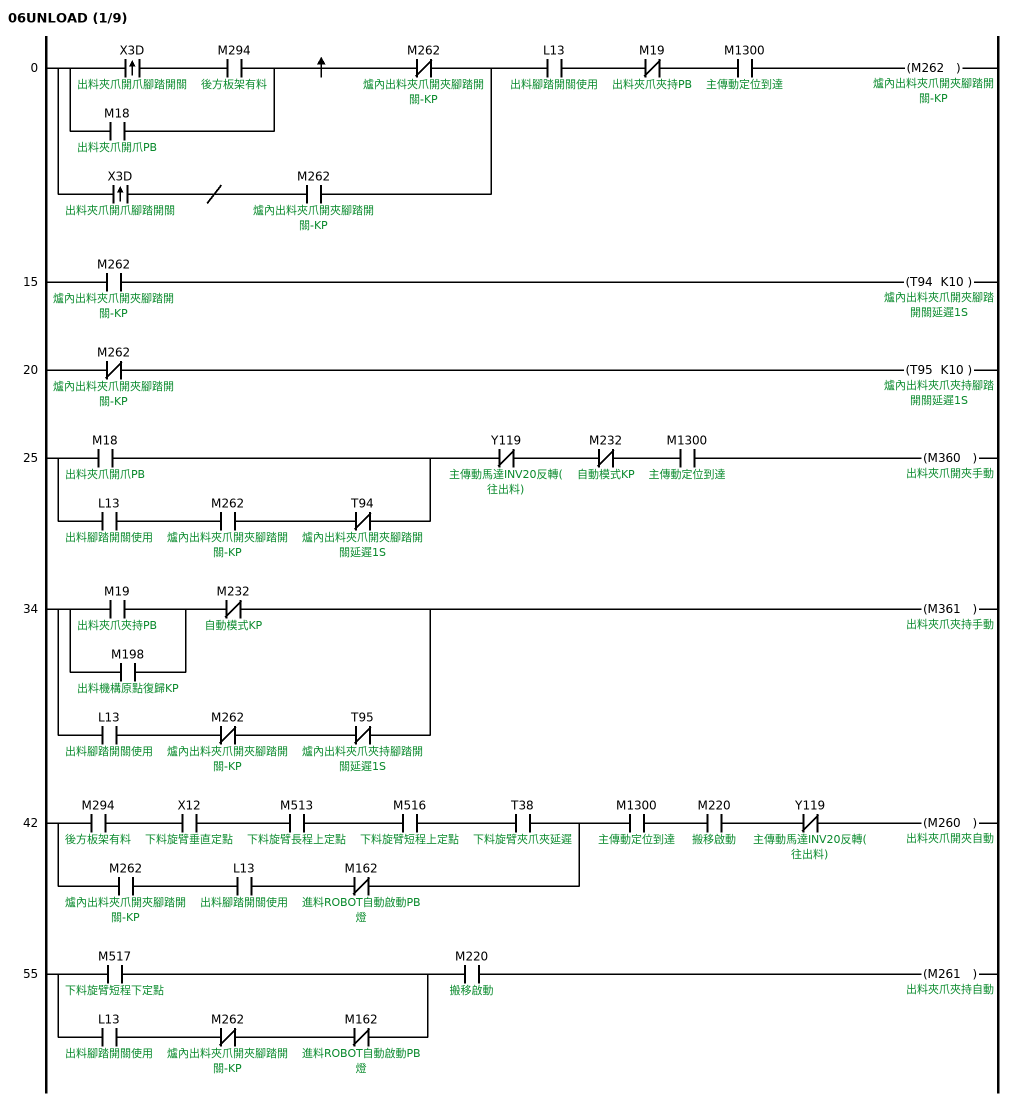
[picture p24: ladder of 06UNLOAD, rungs at steps 0 to 55]
0     LDP     X3D  ; 出料夾爪開爪腳踏開關
      AND     M294  ; 後方板架有料
      OR      M18  ; 出料夾爪開爪PB
      MEP
      ANI     M262  ; 爐內出料夾爪開夾腳踏開關-KP
      LDP     X3D  ; 出料夾爪開爪腳踏開關
      INV
      AND     M262  ; 爐內出料夾爪開夾腳踏開關-KP
      ORB
      AND     L13  ; 出料腳踏開關使用
      ANI     M19  ; 出料夾爪夾持PB
      AND     M1300  ; 主傳動定位到達
      OUT     M262  ; 爐內出料夾爪開夾腳踏開關-KP
15    LD      M262  ; 爐內出料夾爪開夾腳踏開關-KP
      OUT     T94 K10  ; 爐內出料夾爪開夾腳踏開關延遲1S
20    LDI     M262  ; 爐內出料夾爪開夾腳踏開關-KP
      OUT     T95 K10  ; 爐內出料夾爪夾持腳踏開關延遲1S
25    LD      M18  ; 出料夾爪開爪PB
      LD      L13  ; 出料腳踏開關使用
      AND     M262  ; 爐內出料夾爪開夾腳踏開關-KP
      ANI     T94  ; 爐內出料夾爪開夾腳踏開關延遲1S
      ORB
      ANI     Y119  ; 主傳動馬達INV20反轉(往出料)
      ANI     M232  ; 自動模式KP
      AND     M1300  ; 主傳動定位到達
      OUT     M360  ; 出料夾爪開夾手動
34    LD      M19  ; 出料夾爪夾持PB
      OR      M198  ; 出料機構原點復歸KP
      ANI     M232  ; 自動模式KP
      LD      L13  ; 出料腳踏開關使用
      ANI     M262  ; 爐內出料夾爪開夾腳踏開關-KP
      ANI     T95  ; 爐內出料夾爪夾持腳踏開關延遲1S
      ORB
      OUT     M361  ; 出料夾爪夾持手動
42    LD      M294  ; 後方板架有料
      AND     X12  ; 下料旋臂垂直定點
      AND     M513  ; 下料旋臂長程上定點
      AND     M516  ; 下料旋臂短程上定點
      AND     T38  ; 下料旋臂夾爪夾延遲
      LD      M262  ; 爐內出料夾爪開夾腳踏開關-KP
      AND     L13  ; 出料腳踏開關使用
      ANI     M162  ; 進料ROBOT自動啟動PB燈
      ORB
      AND     M1300  ; 主傳動定位到達
      AND     M220  ; 搬移啟動
      ANI     Y119  ; 主傳動馬達INV20反轉(往出料)
      OUT     M260  ; 出料夾爪開夾自動
55    LD      M517  ; 下料旋臂短程下定點
      LD      L13  ; 出料腳踏開關使用
      ANI     M262  ; 爐內出料夾爪開夾腳踏開關-KP
      ANI     M162  ; 進料ROBOT自動啟動PB燈
      ORB
      AND     M220  ; 搬移啟動
      OUT     M261  ; 出料夾爪夾持自動
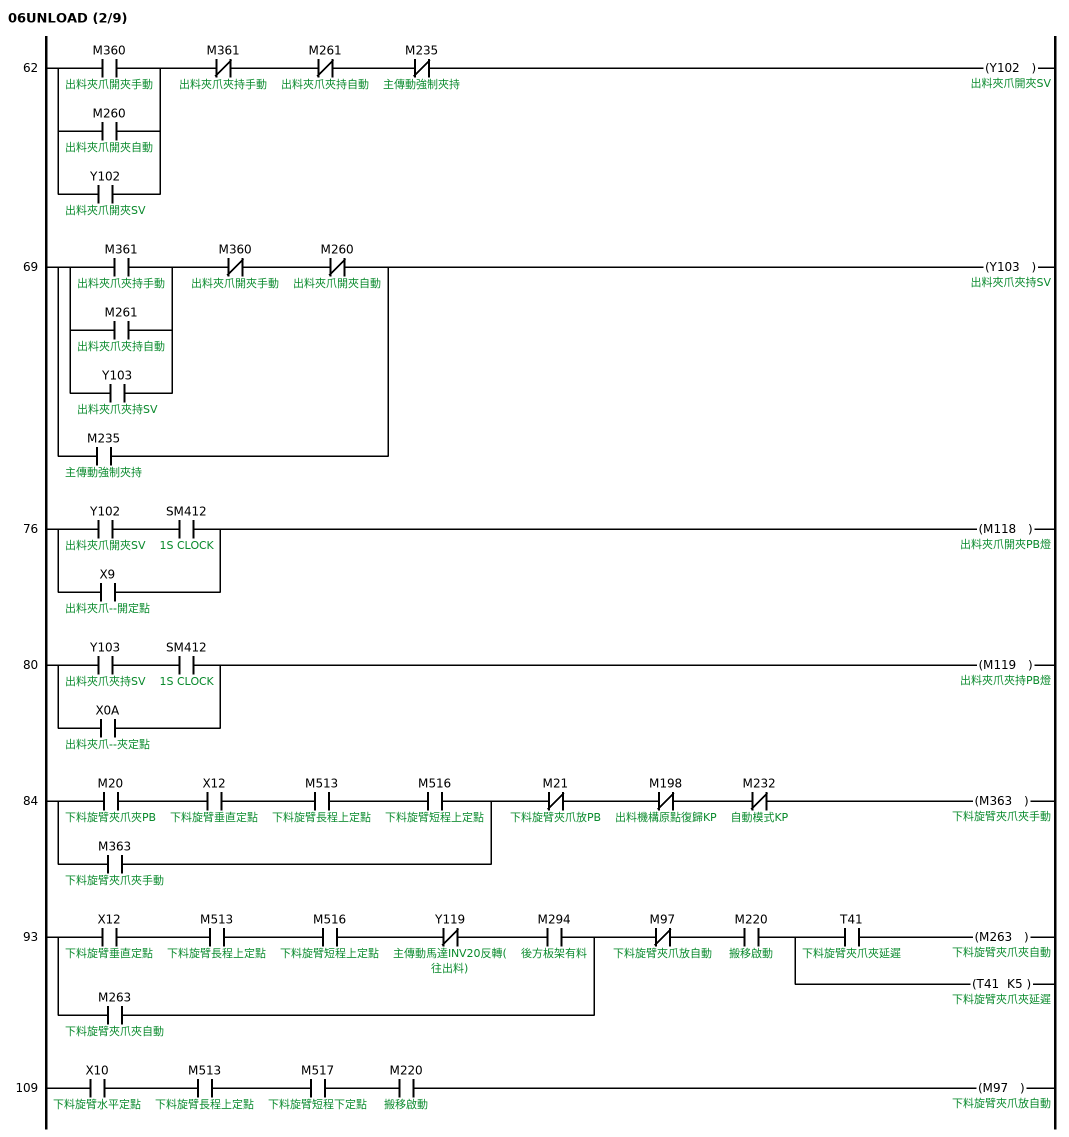
62    LD      M360  ; 出料夾爪開夾手動
      OR      M260  ; 出料夾爪開夾自動
      OR      Y102  ; 出料夾爪開夾SV
      ANI     M361  ; 出料夾爪夾持手動
      ANI     M261  ; 出料夾爪夾持自動
      ANI     M235  ; 主傳動強制夾持
      OUT     Y102  ; 出料夾爪開夾SV
69    LD      M361  ; 出料夾爪夾持手動
      OR      M261  ; 出料夾爪夾持自動
      OR      Y103  ; 出料夾爪夾持SV
      ANI     M360  ; 出料夾爪開夾手動
      ANI     M260  ; 出料夾爪開夾自動
      OR      M235  ; 主傳動強制夾持
      OUT     Y103  ; 出料夾爪夾持SV
76    LD      Y102  ; 出料夾爪開夾SV
      AND     SM412  ; 1S CLOCK
      OR      X9  ; 出料夾爪--開定點
      OUT     M118  ; 出料夾爪開夾PB燈
80    LD      Y103  ; 出料夾爪夾持SV
      AND     SM412  ; 1S CLOCK
      OR      X0A  ; 出料夾爪--夾定點
      OUT     M119  ; 出料夾爪夾持PB燈
84    LD      M20  ; 下料旋臂夾爪夾PB
      AND     X12  ; 下料旋臂垂直定點
      AND     M513  ; 下料旋臂長程上定點
      AND     M516  ; 下料旋臂短程上定點
      OR      M363  ; 下料旋臂夾爪夾手動
      ANI     M21  ; 下料旋臂夾爪放PB
      ANI     M198  ; 出料機構原點復歸KP
      ANI     M232  ; 自動模式KP
      OUT     M363  ; 下料旋臂夾爪夾手動
93    LD      X12  ; 下料旋臂垂直定點
      AND     M513  ; 下料旋臂長程上定點
      AND     M516  ; 下料旋臂短程上定點
      ANI     Y119  ; 主傳動馬達INV20反轉(往出料)
      AND     M294  ; 後方板架有料
      OR      M263  ; 下料旋臂夾爪夾自動
      ANI     M97  ; 下料旋臂夾爪放自動
      AND     M220  ; 搬移啟動
      MPS
      AND     T41  ; 下料旋臂夾爪夾延遲
      OUT     M263  ; 下料旋臂夾爪夾自動
      MPP
      OUT     T41 K5  ; 下料旋臂夾爪夾延遲
109   LD      X10  ; 下料旋臂水平定點
      AND     M513  ; 下料旋臂長程上定點
      AND     M517  ; 下料旋臂短程下定點
      AND     M220  ; 搬移啟動
      OUT     M97  ; 下料旋臂夾爪放自動
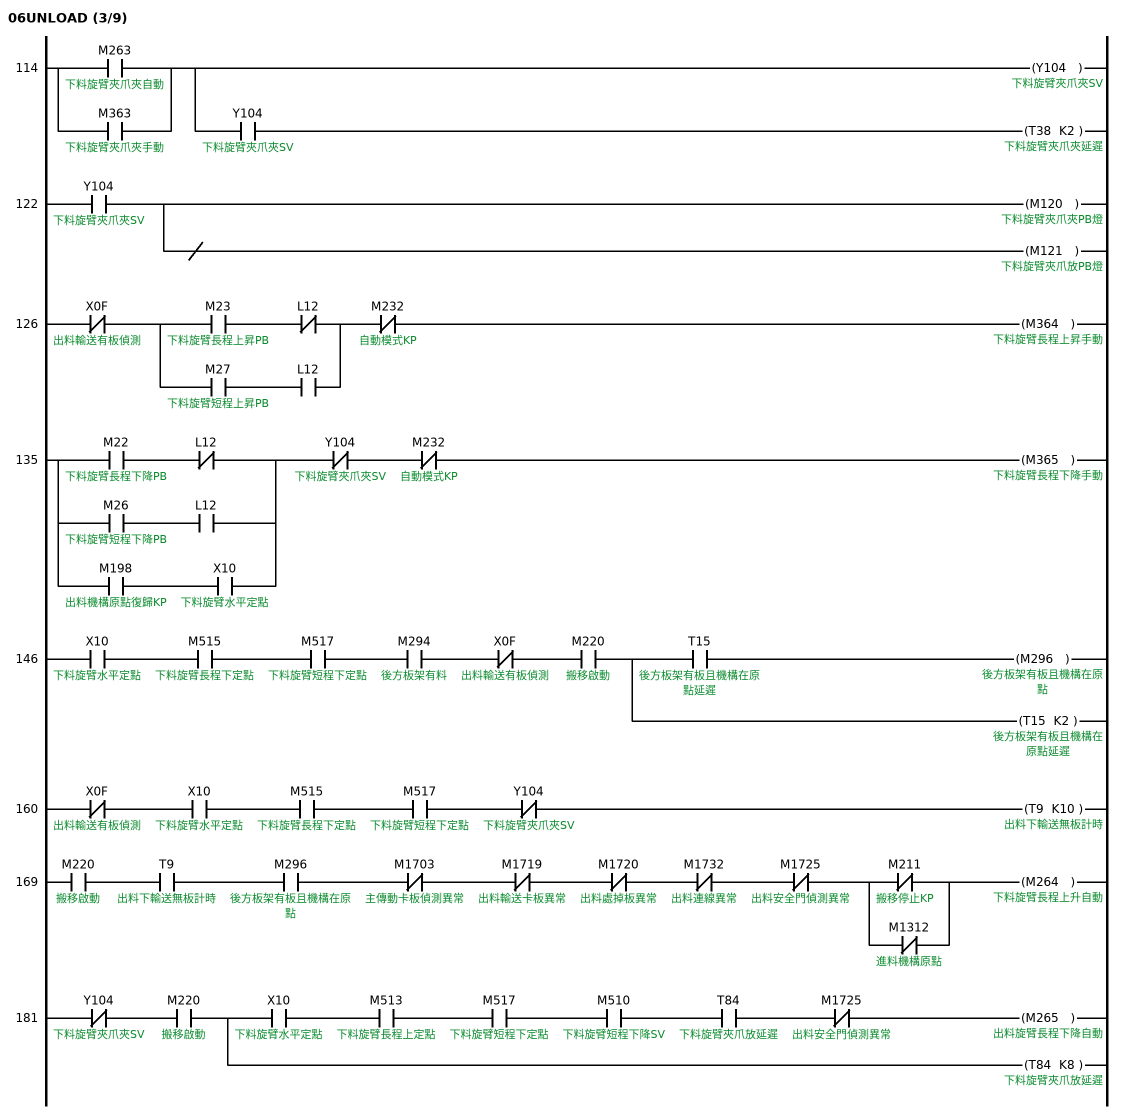
114   LD      M263  ; 下料旋臂夾爪夾自動
      OR      M363  ; 下料旋臂夾爪夾手動
      OUT     Y104  ; 下料旋臂夾爪夾SV
      AND     Y104  ; 下料旋臂夾爪夾SV
      OUT     T38 K2  ; 下料旋臂夾爪夾延遲
122   LD      Y104  ; 下料旋臂夾爪夾SV
      OUT     M120  ; 下料旋臂夾爪夾PB燈
      INV
      OUT     M121  ; 下料旋臂夾爪放PB燈
126   LDI     X0F  ; 出料輸送有板偵測
      LD      M23  ; 下料旋臂長程上昇PB
      ANI     L12
      LD      M27  ; 下料旋臂短程上昇PB
      AND     L12
      ORB
      ANB
      ANI     M232  ; 自動模式KP
      OUT     M364  ; 下料旋臂長程上昇手動
135   LD      M22  ; 下料旋臂長程下降PB
      ANI     L12
      LD      M26  ; 下料旋臂短程下降PB
      AND     L12
      ORB
      LD      M198  ; 出料機構原點復歸KP
      AND     X10  ; 下料旋臂水平定點
      ORB
      ANI     Y104  ; 下料旋臂夾爪夾SV
      ANI     M232  ; 自動模式KP
      OUT     M365  ; 下料旋臂長程下降手動
146   LD      X10  ; 下料旋臂水平定點
      AND     M515  ; 下料旋臂長程下定點
      AND     M517  ; 下料旋臂短程下定點
      AND     M294  ; 後方板架有料
      ANI     X0F  ; 出料輸送有板偵測
      AND     M220  ; 搬移啟動
      MPS
      AND     T15  ; 後方板架有板且機構在原點延遲
      OUT     M296  ; 後方板架有板且機構在原點
      MPP
      OUT     T15 K2  ; 後方板架有板且機構在原點延遲
160   LDI     X0F  ; 出料輸送有板偵測
      AND     X10  ; 下料旋臂水平定點
      AND     M515  ; 下料旋臂長程下定點
      AND     M517  ; 下料旋臂短程下定點
      ANI     Y104  ; 下料旋臂夾爪夾SV
      OUT     T9 K10  ; 出料下輸送無板計時
169   LD      M220  ; 搬移啟動
      AND     T9  ; 出料下輸送無板計時
      AND     M296  ; 後方板架有板且機構在原點
      ANI     M1703  ; 主傳動卡板偵測異常
      ANI     M1719  ; 出料輸送卡板異常
      ANI     M1720  ; 出料處掉板異常
      ANI     M1732  ; 出料連線異常
      ANI     M1725  ; 出料安全門偵測異常
      LDI     M211  ; 搬移停止KP
      ORI     M1312  ; 進料機構原點
      ANB
      OUT     M264  ; 下料旋臂長程上升自動
181   LDI     Y104  ; 下料旋臂夾爪夾SV
      AND     M220  ; 搬移啟動
      MPS
      AND     X10  ; 下料旋臂水平定點
      AND     M513  ; 下料旋臂長程上定點
      AND     M517  ; 下料旋臂短程下定點
      AND     M510  ; 下料旋臂短程下降SV
      AND     T84  ; 下料旋臂夾爪放延遲
      ANI     M1725  ; 出料安全門偵測異常
      OUT     M265  ; 出料旋臂長程下降自動
      MPP
      OUT     T84 K8  ; 下料旋臂夾爪放延遲
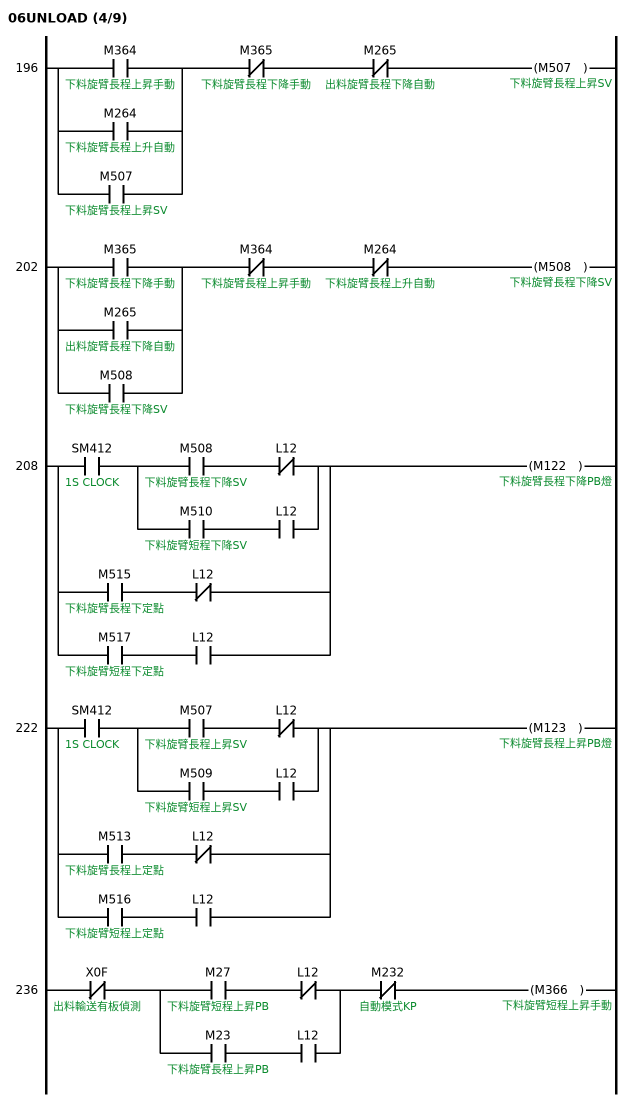
196   LD      M364  ; 下料旋臂長程上昇手動
      OR      M264  ; 下料旋臂長程上升自動
      OR      M507  ; 下料旋臂長程上昇SV
      ANI     M365  ; 下料旋臂長程下降手動
      ANI     M265  ; 出料旋臂長程下降自動
      OUT     M507  ; 下料旋臂長程上昇SV
202   LD      M365  ; 下料旋臂長程下降手動
      OR      M265  ; 出料旋臂長程下降自動
      OR      M508  ; 下料旋臂長程下降SV
      ANI     M364  ; 下料旋臂長程上昇手動
      ANI     M264  ; 下料旋臂長程上升自動
      OUT     M508  ; 下料旋臂長程下降SV
208   LD      SM412  ; 1S CLOCK
      LD      M508  ; 下料旋臂長程下降SV
      ANI     L12
      LD      M510  ; 下料旋臂短程下降SV
      AND     L12
      ORB
      ANB
      LD      M515  ; 下料旋臂長程下定點
      ANI     L12
      ORB
      LD      M517  ; 下料旋臂短程下定點
      AND     L12
      ORB
      OUT     M122  ; 下料旋臂長程下降PB燈
222   LD      SM412  ; 1S CLOCK
      LD      M507  ; 下料旋臂長程上昇SV
      ANI     L12
      LD      M509  ; 下料旋臂短程上昇SV
      AND     L12
      ORB
      ANB
      LD      M513  ; 下料旋臂長程上定點
      ANI     L12
      ORB
      LD      M516  ; 下料旋臂短程上定點
      AND     L12
      ORB
      OUT     M123  ; 下料旋臂長程上昇PB燈
236   LDI     X0F  ; 出料輸送有板偵測
      LD      M27  ; 下料旋臂短程上昇PB
      ANI     L12
      LD      M23  ; 下料旋臂長程上昇PB
      AND     L12
      ORB
      ANB
      ANI     M232  ; 自動模式KP
      OUT     M366  ; 下料旋臂短程上昇手動
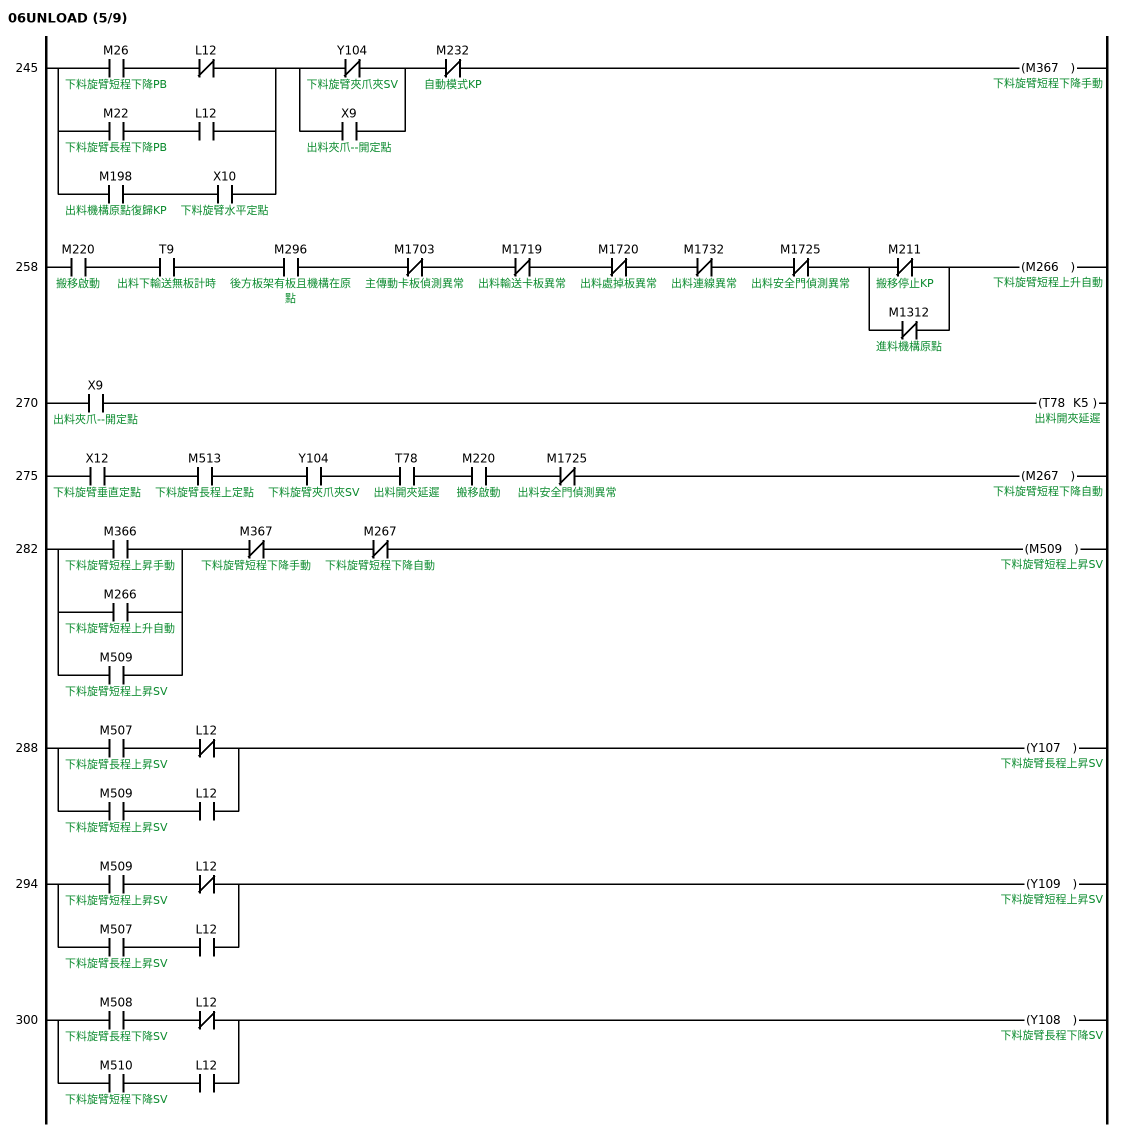
245   LD      M26  ; 下料旋臂短程下降PB
      ANI     L12
      LD      M22  ; 下料旋臂長程下降PB
      AND     L12
      ORB
      LD      M198  ; 出料機構原點復歸KP
      AND     X10  ; 下料旋臂水平定點
      ORB
      LDI     Y104  ; 下料旋臂夾爪夾SV
      OR      X9  ; 出料夾爪--開定點
      ANB
      ANI     M232  ; 自動模式KP
      OUT     M367  ; 下料旋臂短程下降手動
258   LD      M220  ; 搬移啟動
      AND     T9  ; 出料下輸送無板計時
      AND     M296  ; 後方板架有板且機構在原點
      ANI     M1703  ; 主傳動卡板偵測異常
      ANI     M1719  ; 出料輸送卡板異常
      ANI     M1720  ; 出料處掉板異常
      ANI     M1732  ; 出料連線異常
      ANI     M1725  ; 出料安全門偵測異常
      LDI     M211  ; 搬移停止KP
      ORI     M1312  ; 進料機構原點
      ANB
      OUT     M266  ; 下料旋臂短程上升自動
270   LD      X9  ; 出料夾爪--開定點
      OUT     T78 K5  ; 出料開夾延遲
275   LD      X12  ; 下料旋臂垂直定點
      AND     M513  ; 下料旋臂長程上定點
      AND     Y104  ; 下料旋臂夾爪夾SV
      AND     T78  ; 出料開夾延遲
      AND     M220  ; 搬移啟動
      ANI     M1725  ; 出料安全門偵測異常
      OUT     M267  ; 下料旋臂短程下降自動
282   LD      M366  ; 下料旋臂短程上昇手動
      OR      M266  ; 下料旋臂短程上升自動
      OR      M509  ; 下料旋臂短程上昇SV
      ANI     M367  ; 下料旋臂短程下降手動
      ANI     M267  ; 下料旋臂短程下降自動
      OUT     M509  ; 下料旋臂短程上昇SV
288   LD      M507  ; 下料旋臂長程上昇SV
      ANI     L12
      LD      M509  ; 下料旋臂短程上昇SV
      AND     L12
      ORB
      OUT     Y107  ; 下料旋臂長程上昇SV
294   LD      M509  ; 下料旋臂短程上昇SV
      ANI     L12
      LD      M507  ; 下料旋臂長程上昇SV
      AND     L12
      ORB
      OUT     Y109  ; 下料旋臂短程上昇SV
300   LD      M508  ; 下料旋臂長程下降SV
      ANI     L12
      LD      M510  ; 下料旋臂短程下降SV
      AND     L12
      ORB
      OUT     Y108  ; 下料旋臂長程下降SV
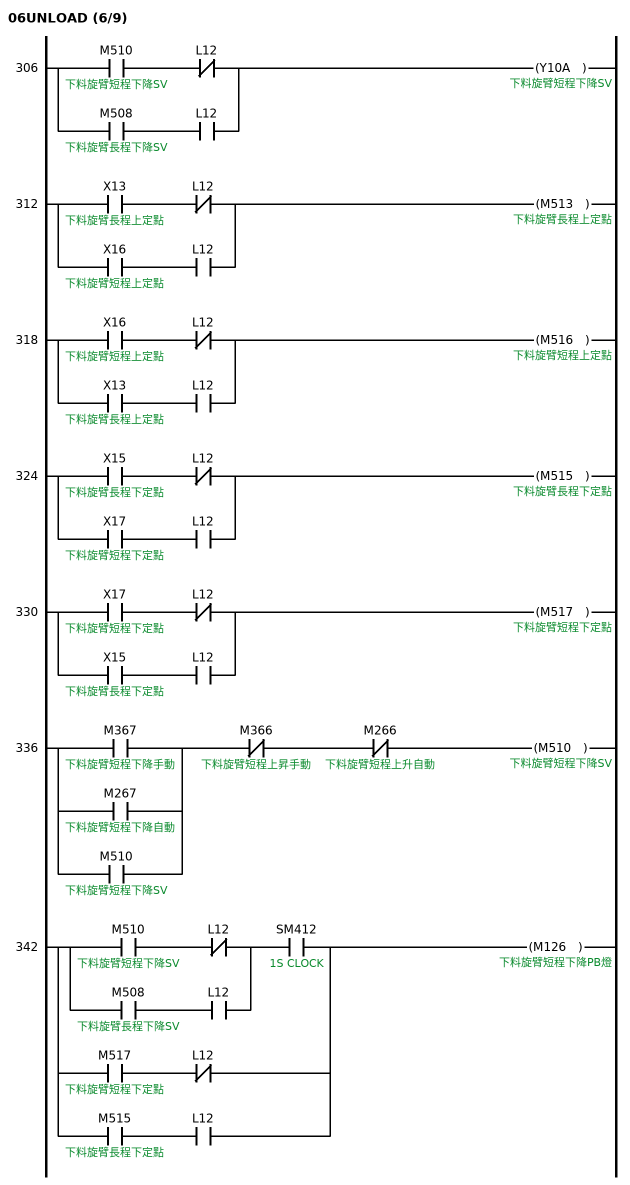
306   LD      M510  ; 下料旋臂短程下降SV
      ANI     L12
      LD      M508  ; 下料旋臂長程下降SV
      AND     L12
      ORB
      OUT     Y10A  ; 下料旋臂短程下降SV
312   LD      X13  ; 下料旋臂長程上定點
      ANI     L12
      LD      X16  ; 下料旋臂短程上定點
      AND     L12
      ORB
      OUT     M513  ; 下料旋臂長程上定點
318   LD      X16  ; 下料旋臂短程上定點
      ANI     L12
      LD      X13  ; 下料旋臂長程上定點
      AND     L12
      ORB
      OUT     M516  ; 下料旋臂短程上定點
324   LD      X15  ; 下料旋臂長程下定點
      ANI     L12
      LD      X17  ; 下料旋臂短程下定點
      AND     L12
      ORB
      OUT     M515  ; 下料旋臂長程下定點
330   LD      X17  ; 下料旋臂短程下定點
      ANI     L12
      LD      X15  ; 下料旋臂長程下定點
      AND     L12
      ORB
      OUT     M517  ; 下料旋臂短程下定點
336   LD      M367  ; 下料旋臂短程下降手動
      OR      M267  ; 下料旋臂短程下降自動
      OR      M510  ; 下料旋臂短程下降SV
      ANI     M366  ; 下料旋臂短程上昇手動
      ANI     M266  ; 下料旋臂短程上升自動
      OUT     M510  ; 下料旋臂短程下降SV
342   LD      M510  ; 下料旋臂短程下降SV
      ANI     L12
      LD      M508  ; 下料旋臂長程下降SV
      AND     L12
      ORB
      AND     SM412  ; 1S CLOCK
      LD      M517  ; 下料旋臂短程下定點
      ANI     L12
      ORB
      LD      M515  ; 下料旋臂長程下定點
      AND     L12
      ORB
      OUT     M126  ; 下料旋臂短程下降PB燈
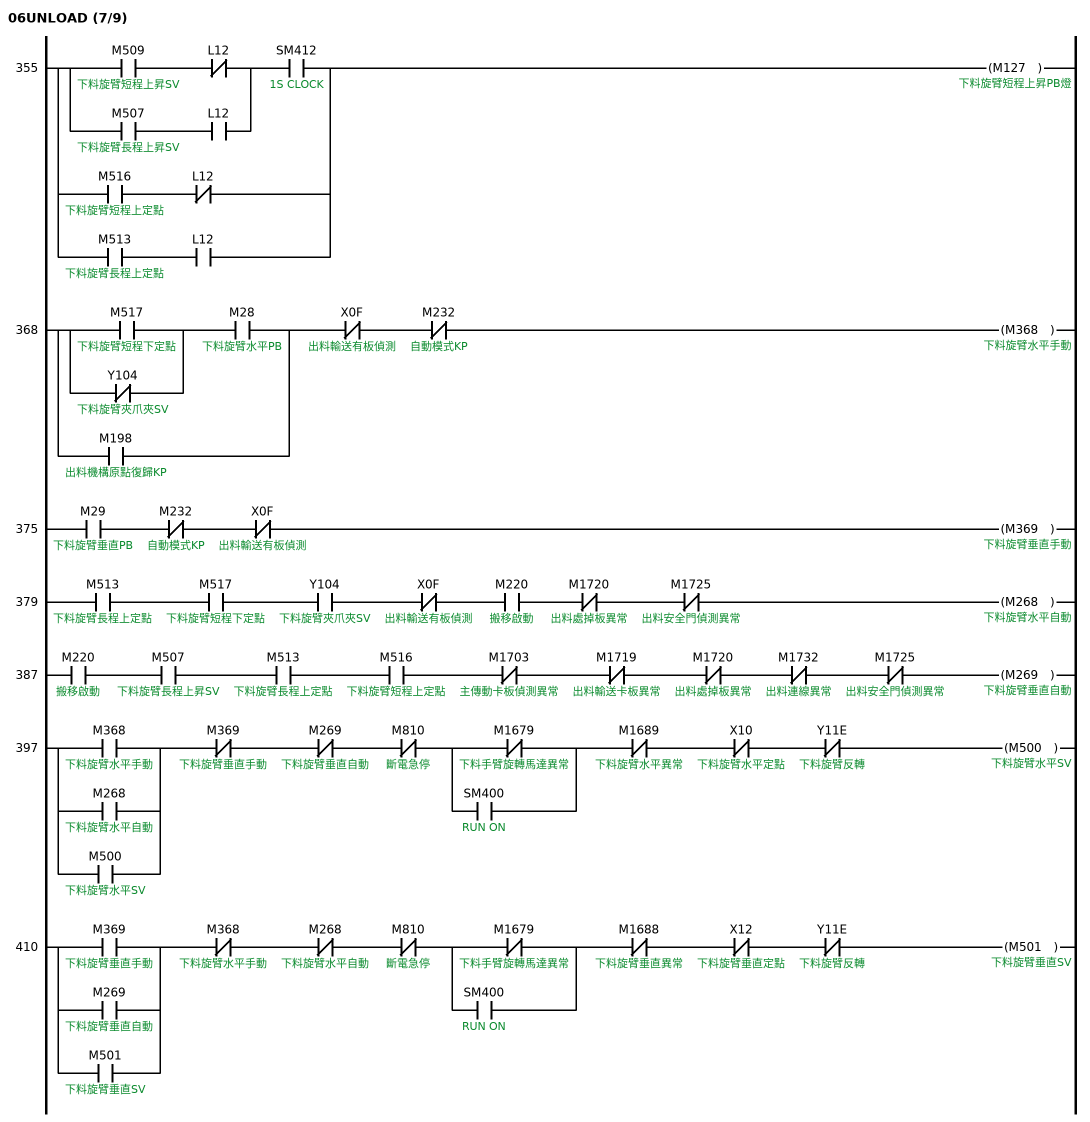
355   LD      M509  ; 下料旋臂短程上昇SV
      ANI     L12
      LD      M507  ; 下料旋臂長程上昇SV
      AND     L12
      ORB
      AND     SM412  ; 1S CLOCK
      LD      M516  ; 下料旋臂短程上定點
      ANI     L12
      ORB
      LD      M513  ; 下料旋臂長程上定點
      AND     L12
      ORB
      OUT     M127  ; 下料旋臂短程上昇PB燈
368   LD      M517  ; 下料旋臂短程下定點
      ORI     Y104  ; 下料旋臂夾爪夾SV
      AND     M28  ; 下料旋臂水平PB
      OR      M198  ; 出料機構原點復歸KP
      ANI     X0F  ; 出料輸送有板偵測
      ANI     M232  ; 自動模式KP
      OUT     M368  ; 下料旋臂水平手動
375   LD      M29  ; 下料旋臂垂直PB
      ANI     M232  ; 自動模式KP
      ANI     X0F  ; 出料輸送有板偵測
      OUT     M369  ; 下料旋臂垂直手動
379   LD      M513  ; 下料旋臂長程上定點
      AND     M517  ; 下料旋臂短程下定點
      AND     Y104  ; 下料旋臂夾爪夾SV
      ANI     X0F  ; 出料輸送有板偵測
      AND     M220  ; 搬移啟動
      ANI     M1720  ; 出料處掉板異常
      ANI     M1725  ; 出料安全門偵測異常
      OUT     M268  ; 下料旋臂水平自動
387   LD      M220  ; 搬移啟動
      AND     M507  ; 下料旋臂長程上昇SV
      AND     M513  ; 下料旋臂長程上定點
      AND     M516  ; 下料旋臂短程上定點
      ANI     M1703  ; 主傳動卡板偵測異常
      ANI     M1719  ; 出料輸送卡板異常
      ANI     M1720  ; 出料處掉板異常
      ANI     M1732  ; 出料連線異常
      ANI     M1725  ; 出料安全門偵測異常
      OUT     M269  ; 下料旋臂垂直自動
397   LD      M368  ; 下料旋臂水平手動
      OR      M268  ; 下料旋臂水平自動
      OR      M500  ; 下料旋臂水平SV
      ANI     M369  ; 下料旋臂垂直手動
      ANI     M269  ; 下料旋臂垂直自動
      ANI     M810  ; 斷電急停
      LDI     M1679  ; 下料手臂旋轉馬達異常
      OR      SM400  ; RUN ON
      ANB
      ANI     M1689  ; 下料旋臂水平異常
      ANI     X10  ; 下料旋臂水平定點
      ANI     Y11E  ; 下料旋臂反轉
      OUT     M500  ; 下料旋臂水平SV
410   LD      M369  ; 下料旋臂垂直手動
      OR      M269  ; 下料旋臂垂直自動
      OR      M501  ; 下料旋臂垂直SV
      ANI     M368  ; 下料旋臂水平手動
      ANI     M268  ; 下料旋臂水平自動
      ANI     M810  ; 斷電急停
      LDI     M1679  ; 下料手臂旋轉馬達異常
      OR      SM400  ; RUN ON
      ANB
      ANI     M1688  ; 下料旋臂垂直異常
      ANI     X12  ; 下料旋臂垂直定點
      ANI     Y11E  ; 下料旋臂反轉
      OUT     M501  ; 下料旋臂垂直SV
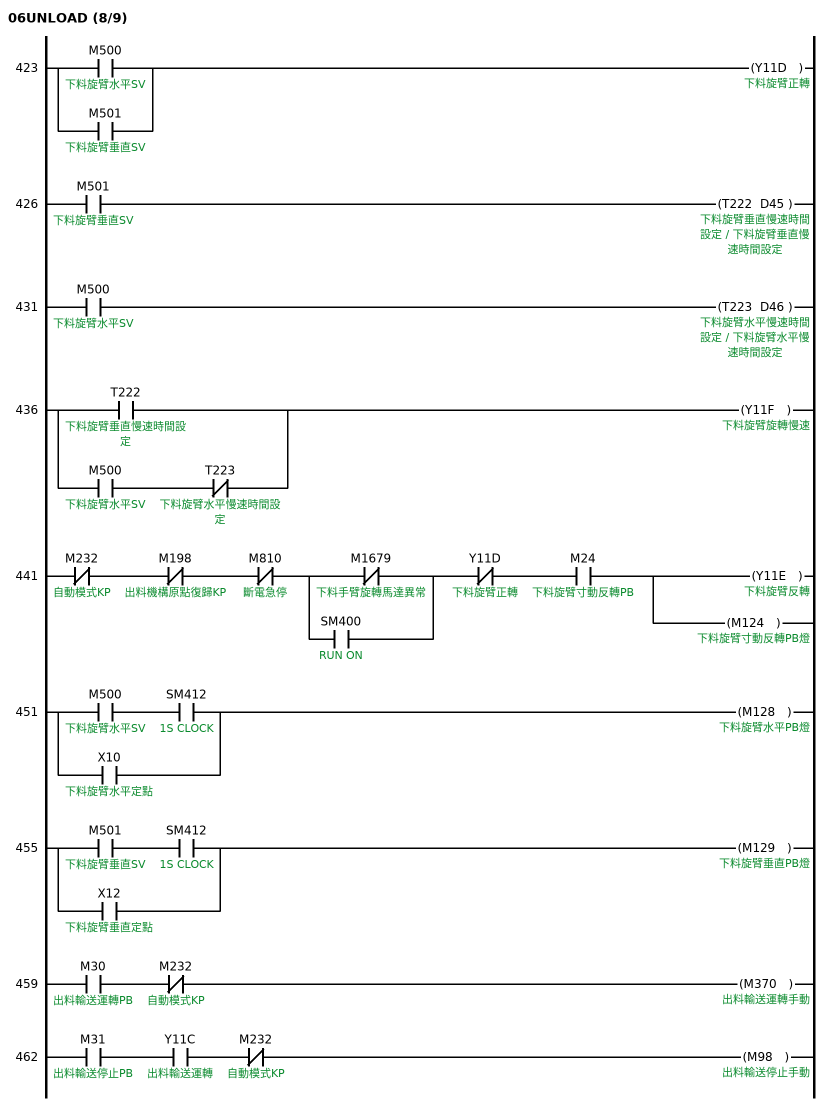
423   LD      M500  ; 下料旋臂水平SV
      OR      M501  ; 下料旋臂垂直SV
      OUT     Y11D  ; 下料旋臂正轉
426   LD      M501  ; 下料旋臂垂直SV
      OUT     T222 D45  ; 下料旋臂垂直慢速時間設定 / 下料旋臂垂直慢速時間設定
431   LD      M500  ; 下料旋臂水平SV
      OUT     T223 D46  ; 下料旋臂水平慢速時間設定 / 下料旋臂水平慢速時間設定
436   LD      T222  ; 下料旋臂垂直慢速時間設定
      LD      M500  ; 下料旋臂水平SV
      ANI     T223  ; 下料旋臂水平慢速時間設定
      ORB
      OUT     Y11F  ; 下料旋臂旋轉慢速
441   LDI     M232  ; 自動模式KP
      ANI     M198  ; 出料機構原點復歸KP
      ANI     M810  ; 斷電急停
      LDI     M1679  ; 下料手臂旋轉馬達異常
      OR      SM400  ; RUN ON
      ANB
      ANI     Y11D  ; 下料旋臂正轉
      AND     M24  ; 下料旋臂寸動反轉PB
      OUT     Y11E  ; 下料旋臂反轉
      OUT     M124  ; 下料旋臂寸動反轉PB燈
451   LD      M500  ; 下料旋臂水平SV
      AND     SM412  ; 1S CLOCK
      OR      X10  ; 下料旋臂水平定點
      OUT     M128  ; 下料旋臂水平PB燈
455   LD      M501  ; 下料旋臂垂直SV
      AND     SM412  ; 1S CLOCK
      OR      X12  ; 下料旋臂垂直定點
      OUT     M129  ; 下料旋臂垂直PB燈
459   LD      M30  ; 出料輸送運轉PB
      ANI     M232  ; 自動模式KP
      OUT     M370  ; 出料輸送運轉手動
462   LD      M31  ; 出料輸送停止PB
      AND     Y11C  ; 出料輸送運轉
      ANI     M232  ; 自動模式KP
      OUT     M98  ; 出料輸送停止手動
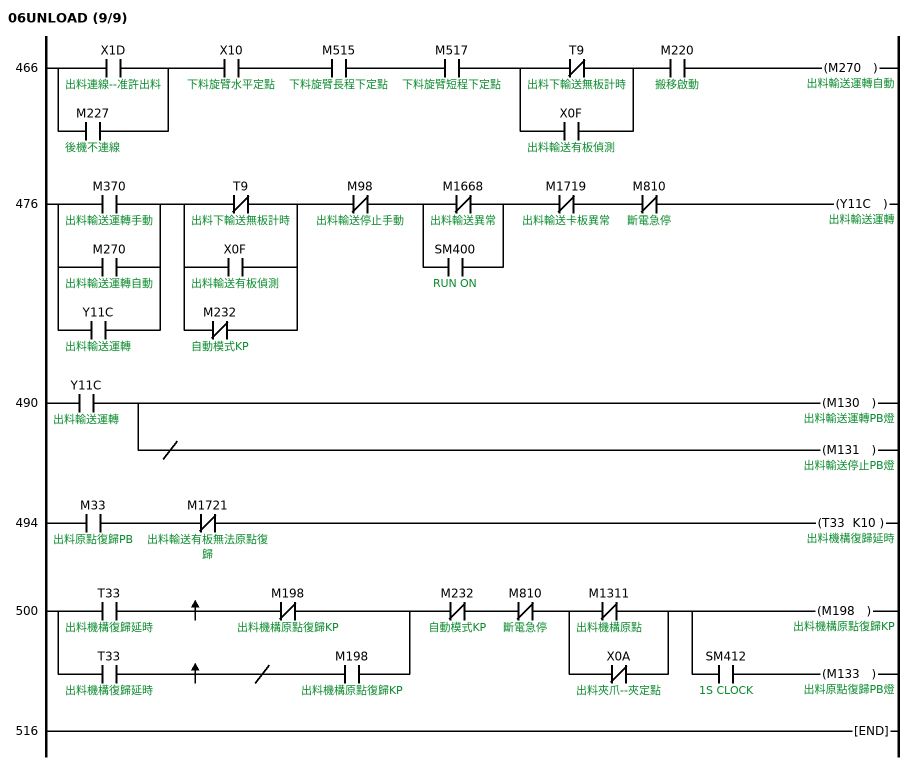
466   LD      X1D  ; 出料連線--准許出料
      OR      M227  ; 後機不連線
      AND     X10  ; 下料旋臂水平定點
      AND     M515  ; 下料旋臂長程下定點
      AND     M517  ; 下料旋臂短程下定點
      LDI     T9  ; 出料下輸送無板計時
      OR      X0F  ; 出料輸送有板偵測
      ANB
      AND     M220  ; 搬移啟動
      OUT     M270  ; 出料輸送運轉自動
476   LD      M370  ; 出料輸送運轉手動
      OR      M270  ; 出料輸送運轉自動
      OR      Y11C  ; 出料輸送運轉
      LDI     T9  ; 出料下輸送無板計時
      OR      X0F  ; 出料輸送有板偵測
      ORI     M232  ; 自動模式KP
      ANB
      ANI     M98  ; 出料輸送停止手動
      LDI     M1668  ; 出料輸送異常
      OR      SM400  ; RUN ON
      ANB
      ANI     M1719  ; 出料輸送卡板異常
      ANI     M810  ; 斷電急停
      OUT     Y11C  ; 出料輸送運轉
490   LD      Y11C  ; 出料輸送運轉
      OUT     M130  ; 出料輸送運轉PB燈
      INV
      OUT     M131  ; 出料輸送停止PB燈
494   LD      M33  ; 出料原點復歸PB
      ANI     M1721  ; 出料輸送有板無法原點復歸
      OUT     T33 K10  ; 出料機構復歸延時
500   LD      T33  ; 出料機構復歸延時
      MEP
      ANI     M198  ; 出料機構原點復歸KP
      LD      T33  ; 出料機構復歸延時
      MEP
      INV
      AND     M198  ; 出料機構原點復歸KP
      ORB
      ANI     M232  ; 自動模式KP
      ANI     M810  ; 斷電急停
      LDI     M1311  ; 出料機構原點
      ORI     X0A  ; 出料夾爪--夾定點
      ANB
      OUT     M198  ; 出料機構原點復歸KP
      AND     SM412  ; 1S CLOCK
      OUT     M133  ; 出料原點復歸PB燈
516   END
END_PROGRAM

PROGRAM 07UNMOVE
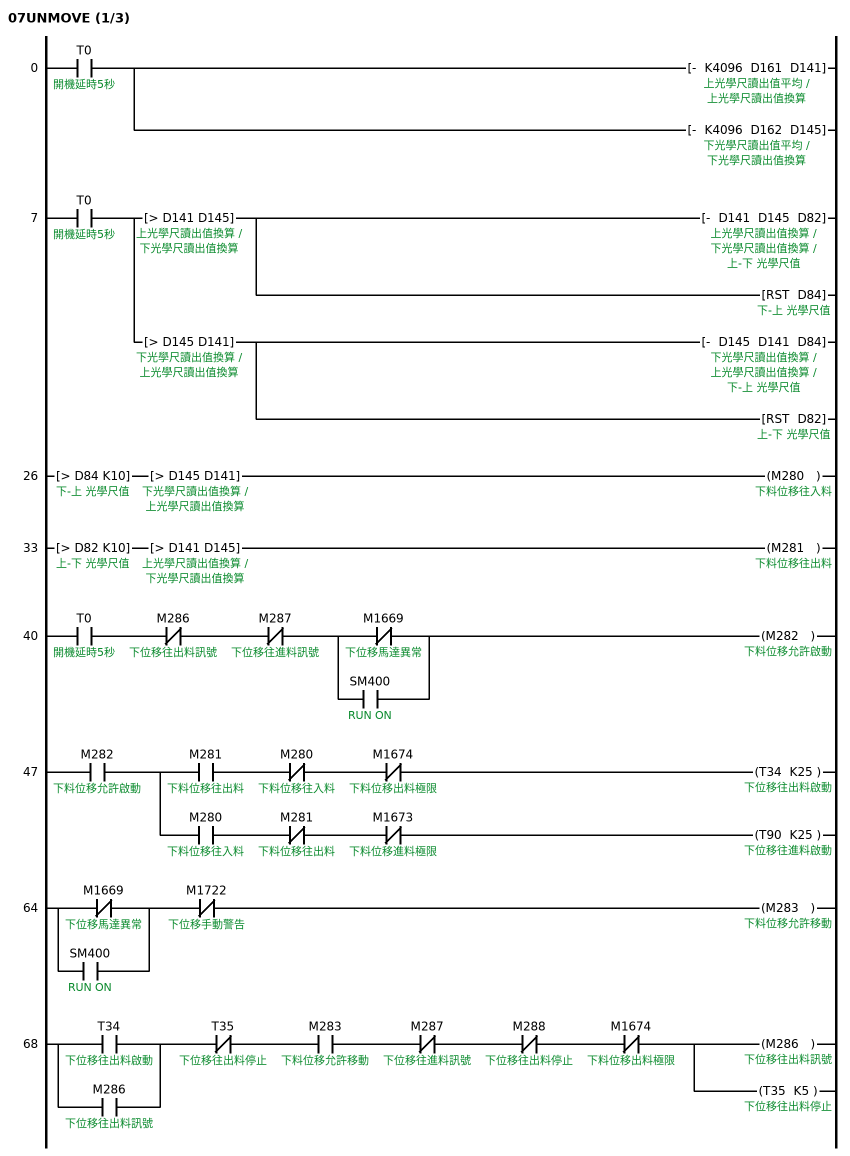
0     LD      T0  ; 開機延時5秒
      -       K4096 D161 D141  ; 上光學尺讀出值平均 / 上光學尺讀出值換算
      -       K4096 D162 D145  ; 下光學尺讀出值平均 / 下光學尺讀出值換算
7     LD      T0  ; 開機延時5秒
      MPS
      AND>    D141 D145  ; 上光學尺讀出值換算 / 下光學尺讀出值換算
      -       D141 D145 D82  ; 上-下 光學尺值
      RST     D84  ; 下-上 光學尺值
      MPP
      AND>    D145 D141  ; 下光學尺讀出值換算 / 上光學尺讀出值換算
      -       D145 D141 D84
      RST     D82  ; 上-下 光學尺值
26    LD>     D84 K10  ; 下-上 光學尺值
      AND>    D145 D141  ; 下光學尺讀出值換算 / 上光學尺讀出值換算
      OUT     M280  ; 下料位移往入料
33    LD>     D82 K10  ; 上-下 光學尺值
      AND>    D141 D145  ; 上光學尺讀出值換算 / 下光學尺讀出值換算
      OUT     M281  ; 下料位移往出料
40    LD      T0  ; 開機延時5秒
      ANI     M286  ; 下位移往出料訊號
      ANI     M287  ; 下位移往進料訊號
      LDI     M1669  ; 下位移馬達異常
      OR      SM400  ; RUN ON
      ANB
      OUT     M282  ; 下料位移允許啟動
47    LD      M282  ; 下料位移允許啟動
      MPS
      AND     M281  ; 下料位移往出料
      ANI     M280  ; 下料位移往入料
      ANI     M1674  ; 下料位移出料極限
      OUT     T34 K25  ; 下位移往出料啟動
      MPP
      AND     M280  ; 下料位移往入料
      ANI     M281  ; 下料位移往出料
      ANI     M1673  ; 下料位移進料極限
      OUT     T90 K25  ; 下位移往進料啟動
64    LDI     M1669  ; 下位移馬達異常
      OR      SM400  ; RUN ON
      ANI     M1722  ; 下位移手動警告
      OUT     M283  ; 下料位移允許移動
68    LD      T34  ; 下位移往出料啟動
      OR      M286  ; 下位移往出料訊號
      ANI     T35  ; 下位移往出料停止
      AND     M283  ; 下料位移允許移動
      ANI     M287  ; 下位移往進料訊號
      ANI     M288  ; 下位移往出料停止
      ANI     M1674  ; 下料位移出料極限
      OUT     M286  ; 下位移往出料訊號
      OUT     T35 K5  ; 下位移往出料停止
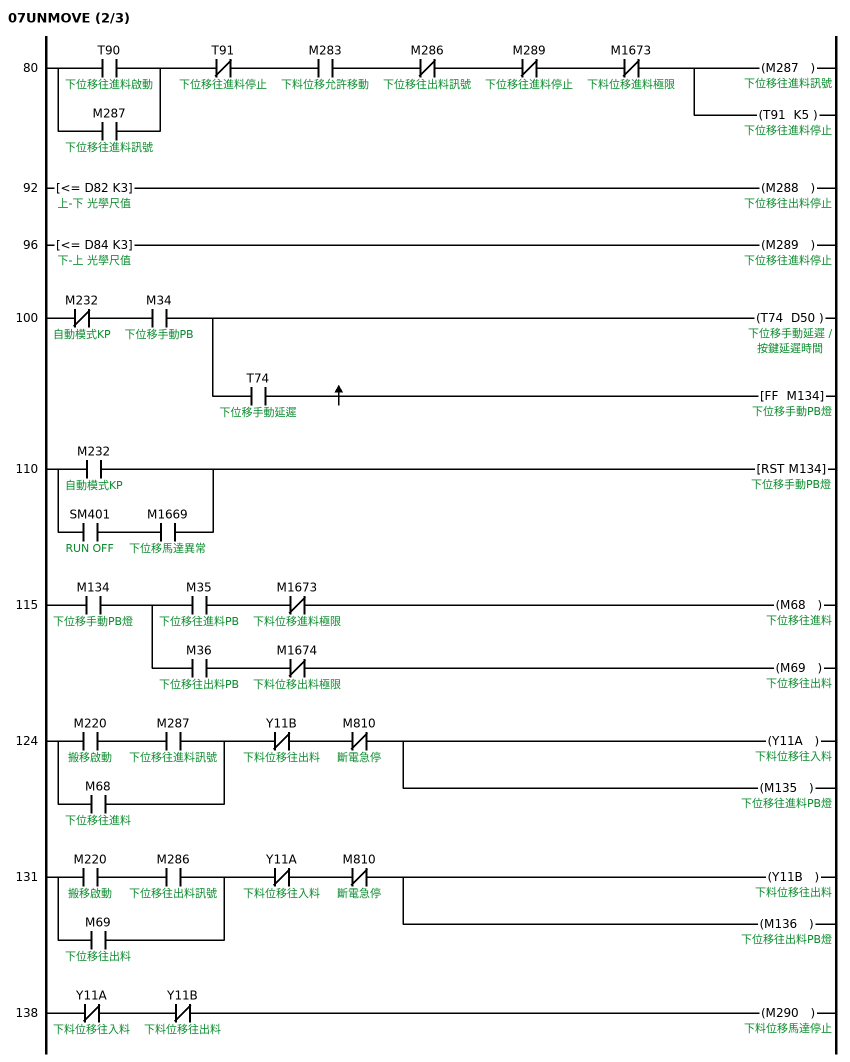
80    LD      T90  ; 下位移往進料啟動
      OR      M287  ; 下位移往進料訊號
      ANI     T91  ; 下位移往進料停止
      AND     M283  ; 下料位移允許移動
      ANI     M286  ; 下位移往出料訊號
      ANI     M289  ; 下位移往進料停止
      ANI     M1673  ; 下料位移進料極限
      OUT     M287  ; 下位移往進料訊號
      OUT     T91 K5  ; 下位移往進料停止
92    LD<=    D82 K3  ; 上-下 光學尺值
      OUT     M288  ; 下位移往出料停止
96    LD<=    D84 K3  ; 下-上 光學尺值
      OUT     M289  ; 下位移往進料停止
100   LDI     M232  ; 自動模式KP
      AND     M34  ; 下位移手動PB
      OUT     T74 D50  ; 下位移手動延遲 / 按鍵延遲時間
      AND     T74  ; 下位移手動延遲
      MEP
      FF      M134  ; 下位移手動PB燈
110   LD      M232  ; 自動模式KP
      LD      SM401  ; RUN OFF
      AND     M1669  ; 下位移馬達異常
      ORB
      RST     M134  ; 下位移手動PB燈
115   LD      M134  ; 下位移手動PB燈
      MPS
      AND     M35  ; 下位移往進料PB
      ANI     M1673  ; 下料位移進料極限
      OUT     M68  ; 下位移往進料
      MPP
      AND     M36  ; 下位移往出料PB
      ANI     M1674  ; 下料位移出料極限
      OUT     M69  ; 下位移往出料
124   LD      M220  ; 搬移啟動
      AND     M287  ; 下位移往進料訊號
      OR      M68  ; 下位移往進料
      ANI     Y11B  ; 下料位移往出料
      ANI     M810  ; 斷電急停
      OUT     Y11A  ; 下料位移往入料
      OUT     M135  ; 下位移往進料PB燈
131   LD      M220  ; 搬移啟動
      AND     M286  ; 下位移往出料訊號
      OR      M69  ; 下位移往出料
      ANI     Y11A  ; 下料位移往入料
      ANI     M810  ; 斷電急停
      OUT     Y11B  ; 下料位移往出料
      OUT     M136  ; 下位移往出料PB燈
138   LDI     Y11A  ; 下料位移往入料
      ANI     Y11B  ; 下料位移往出料
      OUT     M290  ; 下料位移馬達停止
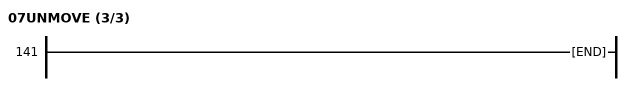
141   END
END_PROGRAM

PROGRAM 08HEATER
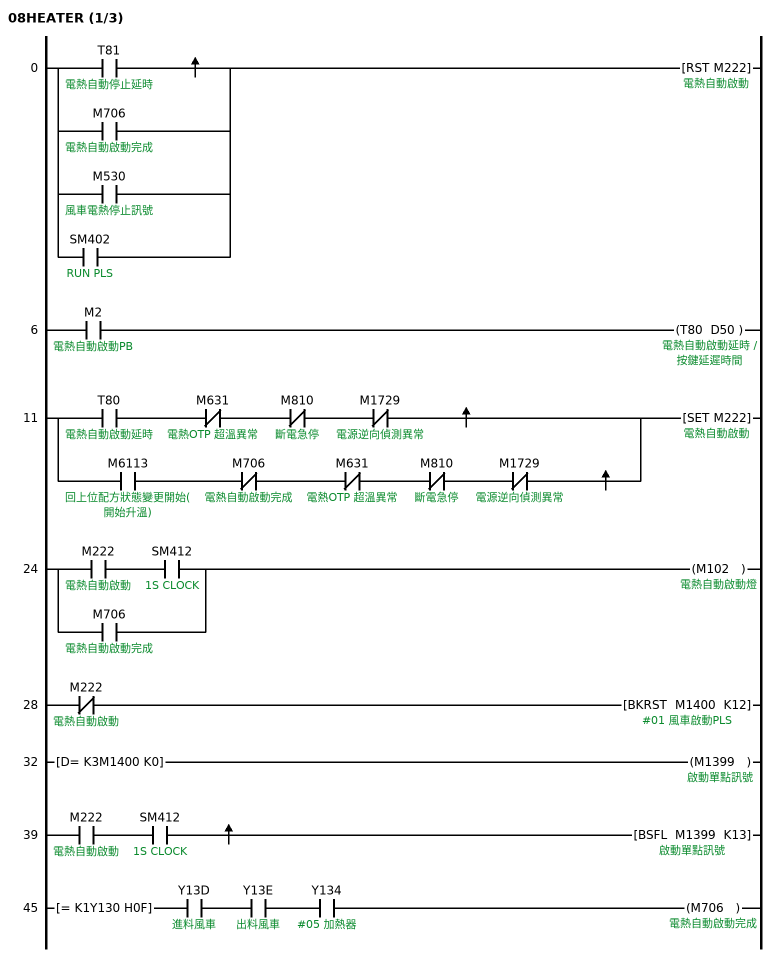
0     LD      T81  ; 電熱自動停止延時
      MEP
      OR      M706  ; 電熱自動啟動完成
      OR      M530  ; 風車電熱停止訊號
      OR      SM402  ; RUN PLS
      RST     M222  ; 電熱自動啟動
6     LD      M2  ; 電熱自動啟動PB
      OUT     T80 D50  ; 電熱自動啟動延時 / 按鍵延遲時間
11    LD      T80  ; 電熱自動啟動延時
      ANI     M631  ; 電熱OTP 超溫異常
      ANI     M810  ; 斷電急停
      ANI     M1729  ; 電源逆向偵測異常
      MEP
      LD      M6113  ; 回上位配方狀態變更開始(開始升溫)
      ANI     M706  ; 電熱自動啟動完成
      ANI     M631  ; 電熱OTP 超溫異常
      ANI     M810  ; 斷電急停
      ANI     M1729  ; 電源逆向偵測異常
      MEP
      ORB
      SET     M222  ; 電熱自動啟動
24    LD      M222  ; 電熱自動啟動
      AND     SM412  ; 1S CLOCK
      OR      M706  ; 電熱自動啟動完成
      OUT     M102  ; 電熱自動啟動燈
28    LDI     M222  ; 電熱自動啟動
      BKRST   M1400 K12  ; #01 風車啟動PLS
32    LDD=    K3M1400 K0  ; #01 風車啟動PLS
      OUT     M1399  ; 啟動單點訊號
39    LD      M222  ; 電熱自動啟動
      AND     SM412  ; 1S CLOCK
      MEP
      BSFL    M1399 K13
45    LD=     K1Y130 H0F  ; #01 加熱器
      AND     Y13D  ; 進料風車
      AND     Y13E  ; 出料風車
      AND     Y134  ; #05 加熱器
      OUT     M706  ; 電熱自動啟動完成
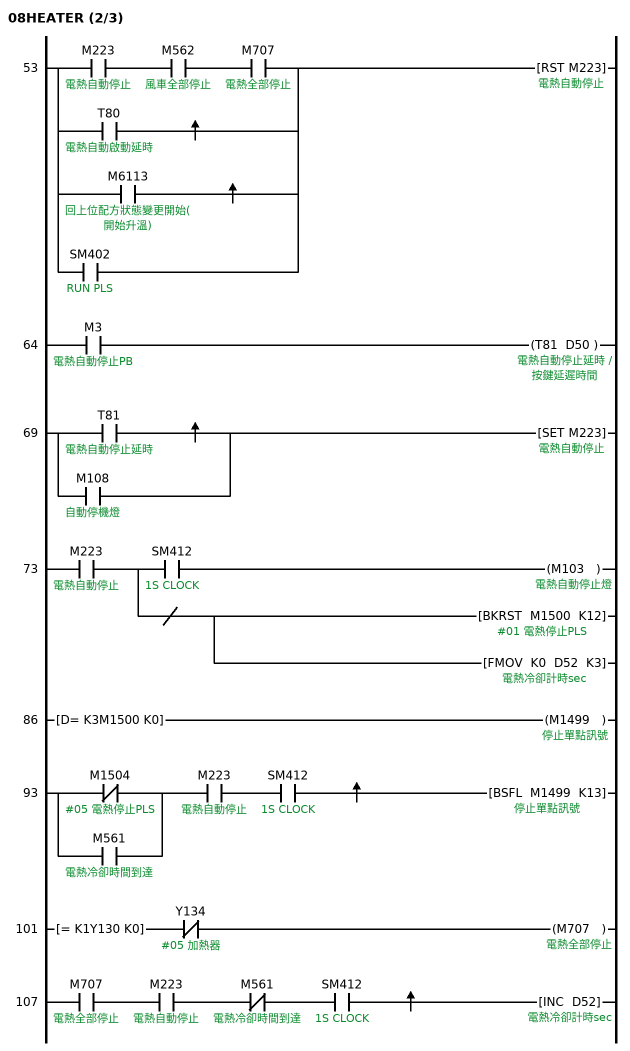
53    LD      M223  ; 電熱自動停止
      AND     M562  ; 風車全部停止
      AND     M707  ; 電熱全部停止
      LD      T80  ; 電熱自動啟動延時
      MEP
      ORB
      LD      M6113  ; 回上位配方狀態變更開始(開始升溫)
      MEP
      ORB
      OR      SM402  ; RUN PLS
      RST     M223  ; 電熱自動停止
64    LD      M3  ; 電熱自動停止PB
      OUT     T81 D50  ; 電熱自動停止延時 / 按鍵延遲時間
69    LD      T81  ; 電熱自動停止延時
      MEP
      OR      M108  ; 自動停機燈
      SET     M223  ; 電熱自動停止
73    LD      M223  ; 電熱自動停止
      MPS
      AND     SM412  ; 1S CLOCK
      OUT     M103  ; 電熱自動停止燈
      MPP
      INV
      BKRST   M1500 K12  ; #01 電熱停止PLS
      FMOV    K0 D52 K3  ; 電熱冷卻計時sec
86    LDD=    K3M1500 K0  ; #01 電熱停止PLS
      OUT     M1499  ; 停止單點訊號
93    LDI     M1504  ; #05 電熱停止PLS
      OR      M561  ; 電熱冷卻時間到達
      AND     M223  ; 電熱自動停止
      AND     SM412  ; 1S CLOCK
      MEP
      BSFL    M1499 K13
101   LD=     K1Y130 K0  ; #01 加熱器
      ANI     Y134  ; #05 加熱器
      OUT     M707  ; 電熱全部停止
107   LD      M707  ; 電熱全部停止
      AND     M223  ; 電熱自動停止
      ANI     M561  ; 電熱冷卻時間到達
      AND     SM412  ; 1S CLOCK
      MEP
      INC     D52
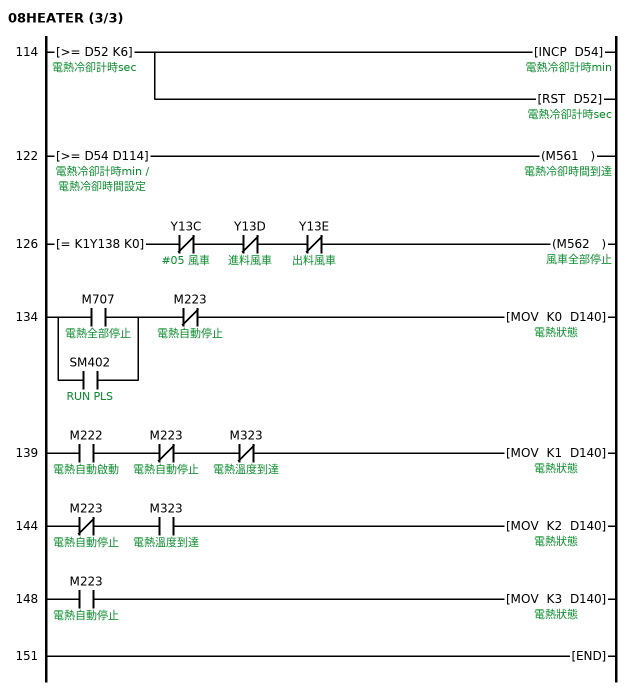
114   LD>=    D52 K6  ; 電熱冷卻計時sec
      INCP    D54  ; 電熱冷卻計時min
      RST     D52  ; 電熱冷卻計時sec
122   LD>=    D54 D114  ; 電熱冷卻計時min / 電熱冷卻時間設定
      OUT     M561  ; 電熱冷卻時間到達
126   LD=     K1Y138 K0  ; #01 風車
      ANI     Y13C  ; #05 風車
      ANI     Y13D  ; 進料風車
      ANI     Y13E  ; 出料風車
      OUT     M562  ; 風車全部停止
134   LD      M707  ; 電熱全部停止
      OR      SM402  ; RUN PLS
      ANI     M223  ; 電熱自動停止
      MOV     K0 D140  ; 電熱狀態
139   LD      M222  ; 電熱自動啟動
      ANI     M223  ; 電熱自動停止
      ANI     M323  ; 電熱溫度到達
      MOV     K1 D140
144   LDI     M223  ; 電熱自動停止
      AND     M323  ; 電熱溫度到達
      MOV     K2 D140
148   LD      M223  ; 電熱自動停止
      MOV     K3 D140
151   END
END_PROGRAM

PROGRAM 09BLOWER
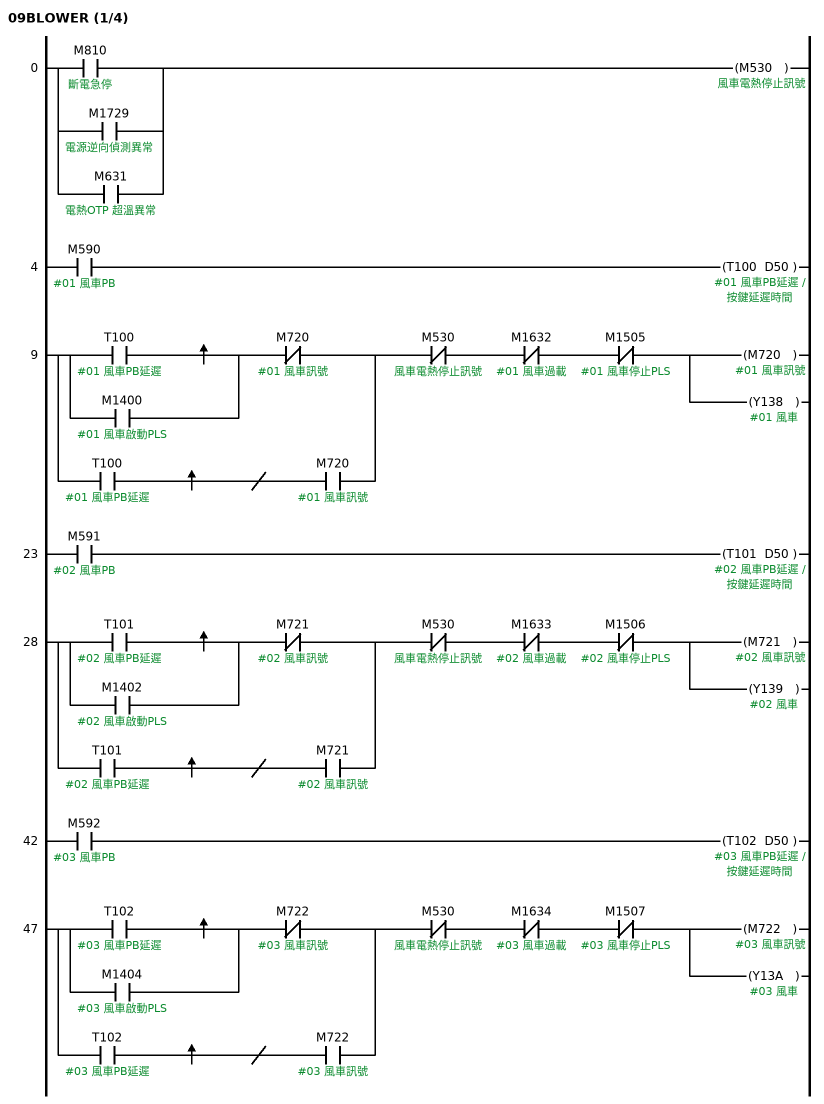
0     LD      M810  ; 斷電急停
      OR      M1729  ; 電源逆向偵測異常
      OR      M631  ; 電熱OTP 超溫異常
      OUT     M530  ; 風車電熱停止訊號
4     LD      M590  ; #01 風車PB
      OUT     T100 D50  ; #01 風車PB延遲 / 按鍵延遲時間
9     LD      T100  ; #01 風車PB延遲
      MEP
      OR      M1400  ; #01 風車啟動PLS
      ANI     M720  ; #01 風車訊號
      LD      T100  ; #01 風車PB延遲
      MEP
      INV
      AND     M720  ; #01 風車訊號
      ORB
      ANI     M530  ; 風車電熱停止訊號
      ANI     M1632  ; #01 風車過載
      ANI     M1505  ; #01 風車停止PLS
      OUT     M720  ; #01 風車訊號
      OUT     Y138  ; #01 風車
23    LD      M591  ; #02 風車PB
      OUT     T101 D50  ; #02 風車PB延遲 / 按鍵延遲時間
28    LD      T101  ; #02 風車PB延遲
      MEP
      OR      M1402  ; #02 風車啟動PLS
      ANI     M721  ; #02 風車訊號
      LD      T101  ; #02 風車PB延遲
      MEP
      INV
      AND     M721  ; #02 風車訊號
      ORB
      ANI     M530  ; 風車電熱停止訊號
      ANI     M1633  ; #02 風車過載
      ANI     M1506  ; #02 風車停止PLS
      OUT     M721  ; #02 風車訊號
      OUT     Y139  ; #02 風車
42    LD      M592  ; #03 風車PB
      OUT     T102 D50  ; #03 風車PB延遲 / 按鍵延遲時間
47    LD      T102  ; #03 風車PB延遲
      MEP
      OR      M1404  ; #03 風車啟動PLS
      ANI     M722  ; #03 風車訊號
      LD      T102  ; #03 風車PB延遲
      MEP
      INV
      AND     M722  ; #03 風車訊號
      ORB
      ANI     M530  ; 風車電熱停止訊號
      ANI     M1634  ; #03 風車過載
      ANI     M1507  ; #03 風車停止PLS
      OUT     M722  ; #03 風車訊號
      OUT     Y13A  ; #03 風車
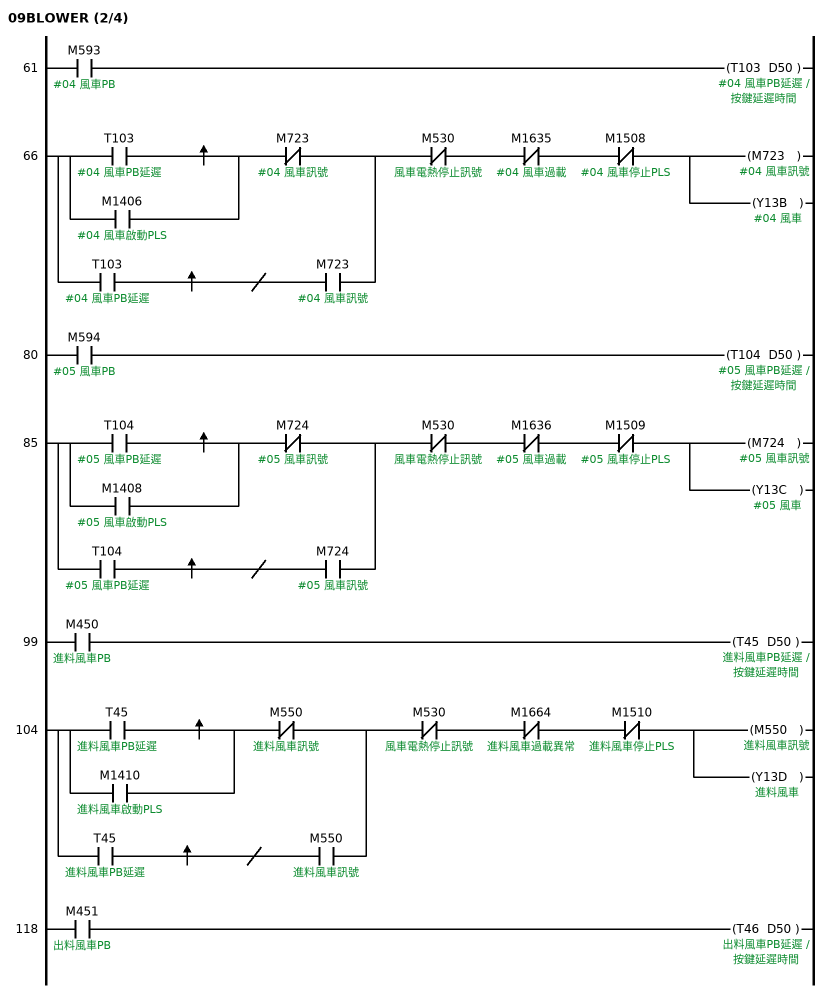
61    LD      M593  ; #04 風車PB
      OUT     T103 D50  ; #04 風車PB延遲 / 按鍵延遲時間
66    LD      T103  ; #04 風車PB延遲
      MEP
      OR      M1406  ; #04 風車啟動PLS
      ANI     M723  ; #04 風車訊號
      LD      T103  ; #04 風車PB延遲
      MEP
      INV
      AND     M723  ; #04 風車訊號
      ORB
      ANI     M530  ; 風車電熱停止訊號
      ANI     M1635  ; #04 風車過載
      ANI     M1508  ; #04 風車停止PLS
      OUT     M723  ; #04 風車訊號
      OUT     Y13B  ; #04 風車
80    LD      M594  ; #05 風車PB
      OUT     T104 D50  ; #05 風車PB延遲 / 按鍵延遲時間
85    LD      T104  ; #05 風車PB延遲
      MEP
      OR      M1408  ; #05 風車啟動PLS
      ANI     M724  ; #05 風車訊號
      LD      T104  ; #05 風車PB延遲
      MEP
      INV
      AND     M724  ; #05 風車訊號
      ORB
      ANI     M530  ; 風車電熱停止訊號
      ANI     M1636  ; #05 風車過載
      ANI     M1509  ; #05 風車停止PLS
      OUT     M724  ; #05 風車訊號
      OUT     Y13C  ; #05 風車
99    LD      M450  ; 進料風車PB
      OUT     T45 D50  ; 進料風車PB延遲 / 按鍵延遲時間
104   LD      T45  ; 進料風車PB延遲
      MEP
      OR      M1410  ; 進料風車啟動PLS
      ANI     M550  ; 進料風車訊號
      LD      T45  ; 進料風車PB延遲
      MEP
      INV
      AND     M550  ; 進料風車訊號
      ORB
      ANI     M530  ; 風車電熱停止訊號
      ANI     M1664  ; 進料風車過載異常
      ANI     M1510  ; 進料風車停止PLS
      OUT     M550  ; 進料風車訊號
      OUT     Y13D  ; 進料風車
118   LD      M451  ; 出料風車PB
      OUT     T46 D50  ; 出料風車PB延遲 / 按鍵延遲時間
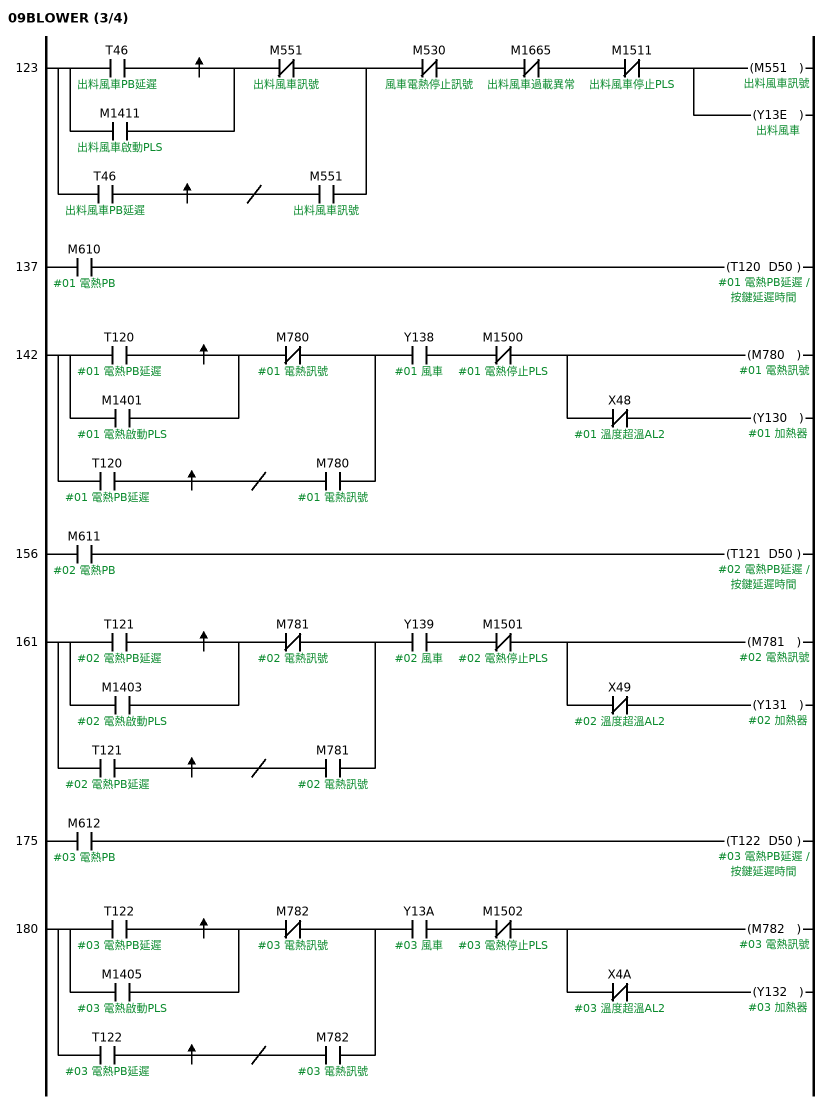
123   LD      T46  ; 出料風車PB延遲
      MEP
      OR      M1411  ; 出料風車啟動PLS
      ANI     M551  ; 出料風車訊號
      LD      T46  ; 出料風車PB延遲
      MEP
      INV
      AND     M551  ; 出料風車訊號
      ORB
      ANI     M530  ; 風車電熱停止訊號
      ANI     M1665  ; 出料風車過載異常
      ANI     M1511  ; 出料風車停止PLS
      OUT     M551  ; 出料風車訊號
      OUT     Y13E  ; 出料風車
137   LD      M610  ; #01 電熱PB
      OUT     T120 D50  ; #01 電熱PB延遲 / 按鍵延遲時間
142   LD      T120  ; #01 電熱PB延遲
      MEP
      OR      M1401  ; #01 電熱啟動PLS
      ANI     M780  ; #01 電熱訊號
      LD      T120  ; #01 電熱PB延遲
      MEP
      INV
      AND     M780  ; #01 電熱訊號
      ORB
      AND     Y138  ; #01 風車
      ANI     M1500  ; #01 電熱停止PLS
      OUT     M780  ; #01 電熱訊號
      ANI     X48  ; #01 溫度超溫AL2
      OUT     Y130  ; #01 加熱器
156   LD      M611  ; #02 電熱PB
      OUT     T121 D50  ; #02 電熱PB延遲 / 按鍵延遲時間
161   LD      T121  ; #02 電熱PB延遲
      MEP
      OR      M1403  ; #02 電熱啟動PLS
      ANI     M781  ; #02 電熱訊號
      LD      T121  ; #02 電熱PB延遲
      MEP
      INV
      AND     M781  ; #02 電熱訊號
      ORB
      AND     Y139  ; #02 風車
      ANI     M1501  ; #02 電熱停止PLS
      OUT     M781  ; #02 電熱訊號
      ANI     X49  ; #02 溫度超溫AL2
      OUT     Y131  ; #02 加熱器
175   LD      M612  ; #03 電熱PB
      OUT     T122 D50  ; #03 電熱PB延遲 / 按鍵延遲時間
180   LD      T122  ; #03 電熱PB延遲
      MEP
      OR      M1405  ; #03 電熱啟動PLS
      ANI     M782  ; #03 電熱訊號
      LD      T122  ; #03 電熱PB延遲
      MEP
      INV
      AND     M782  ; #03 電熱訊號
      ORB
      AND     Y13A  ; #03 風車
      ANI     M1502  ; #03 電熱停止PLS
      OUT     M782  ; #03 電熱訊號
      ANI     X4A  ; #03 溫度超溫AL2
      OUT     Y132  ; #03 加熱器
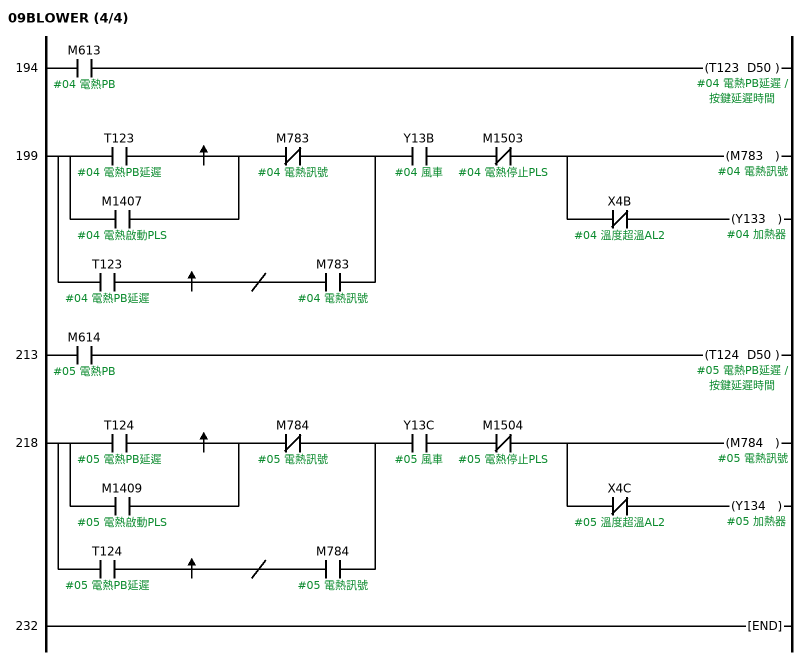
194   LD      M613  ; #04 電熱PB
      OUT     T123 D50  ; #04 電熱PB延遲 / 按鍵延遲時間
199   LD      T123  ; #04 電熱PB延遲
      MEP
      OR      M1407  ; #04 電熱啟動PLS
      ANI     M783  ; #04 電熱訊號
      LD      T123  ; #04 電熱PB延遲
      MEP
      INV
      AND     M783  ; #04 電熱訊號
      ORB
      AND     Y13B  ; #04 風車
      ANI     M1503  ; #04 電熱停止PLS
      OUT     M783  ; #04 電熱訊號
      ANI     X4B  ; #04 溫度超溫AL2
      OUT     Y133  ; #04 加熱器
213   LD      M614  ; #05 電熱PB
      OUT     T124 D50  ; #05 電熱PB延遲 / 按鍵延遲時間
218   LD      T124  ; #05 電熱PB延遲
      MEP
      OR      M1409  ; #05 電熱啟動PLS
      ANI     M784  ; #05 電熱訊號
      LD      T124  ; #05 電熱PB延遲
      MEP
      INV
      AND     M784  ; #05 電熱訊號
      ORB
      AND     Y13C  ; #05 風車
      ANI     M1504  ; #05 電熱停止PLS
      OUT     M784  ; #05 電熱訊號
      ANI     X4C  ; #05 溫度超溫AL2
      OUT     Y134  ; #05 加熱器
232   END
END_PROGRAM

PROGRAM 10YIELD
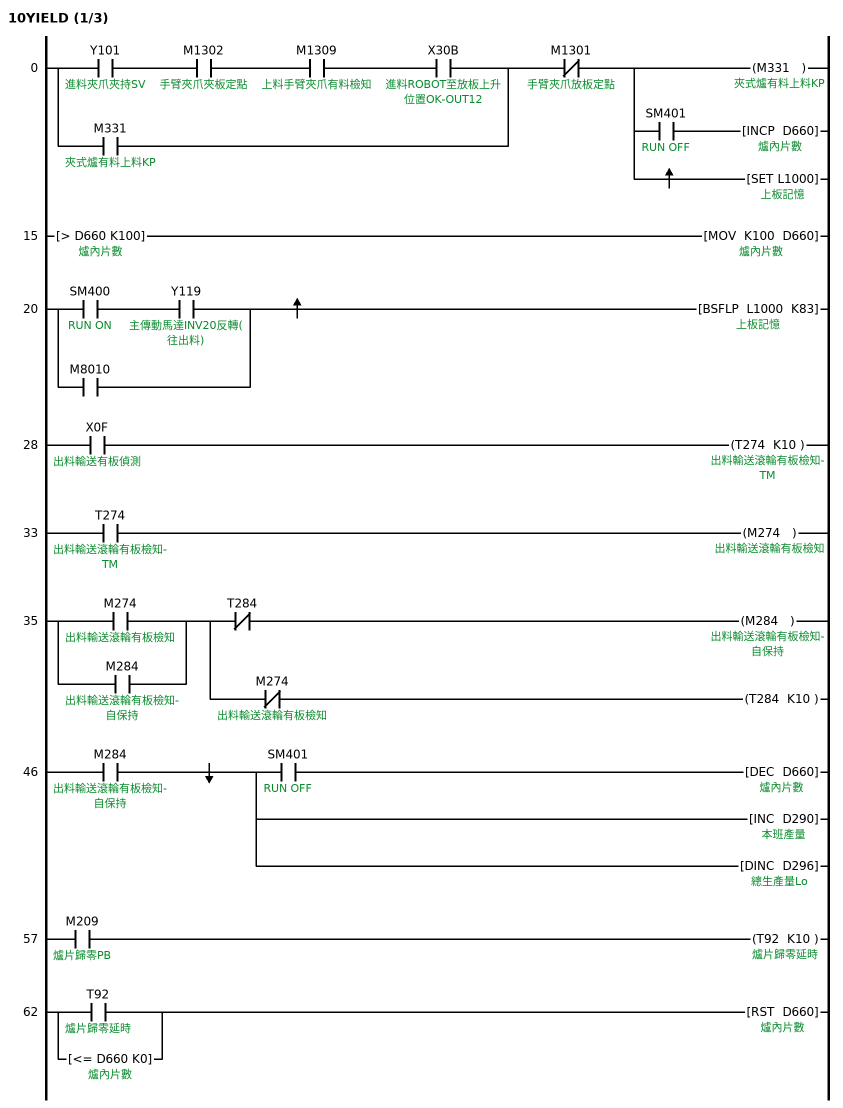
0     LD      Y101  ; 進料夾爪夾持SV
      AND     M1302  ; 手臂夾爪夾板定點
      AND     M1309  ; 上料手臂夾爪有料檢知
      AND     X30B  ; 進料ROBOT至放板上升位置OK-OUT12
      OR      M331  ; 夾式爐有料上料KP
      ANI     M1301  ; 手臂夾爪放板定點
      OUT     M331  ; 夾式爐有料上料KP
      MPS
      AND     SM401  ; RUN OFF
      INCP    D660  ; 爐內片數
      MPP
      MEP
      SET     L1000  ; 上板記憶
15    LD>     D660 K100  ; 爐內片數
      MOV     K100 D660
20    LD      SM400  ; RUN ON
      AND     Y119  ; 主傳動馬達INV20反轉(往出料)
      OR      M8010
      MEP
      BSFLP   L1000 K83
28    LD      X0F  ; 出料輸送有板偵測
      OUT     T274 K10  ; 出料輸送滾輪有板檢知-TM
33    LD      T274  ; 出料輸送滾輪有板檢知-TM
      OUT     M274  ; 出料輸送滾輪有板檢知
35    LD      M274  ; 出料輸送滾輪有板檢知
      OR      M284  ; 出料輸送滾輪有板檢知-自保持
      MPS
      ANI     T284
      OUT     M284  ; 出料輸送滾輪有板檢知-自保持
      MPP
      ANI     M274  ; 出料輸送滾輪有板檢知
      OUT     T284 K10
46    LD      M284  ; 出料輸送滾輪有板檢知-自保持
      MEF
      MPS
      AND     SM401  ; RUN OFF
      DEC     D660
      MPP
      INC     D290  ; 本班產量
      DINC    D296  ; 總生產量Lo
57    LD      M209  ; 爐片歸零PB
      OUT     T92 K10  ; 爐片歸零延時
62    LD      T92  ; 爐片歸零延時
      OR<=    D660 K0  ; 爐內片數
      RST     D660  ; 爐內片數
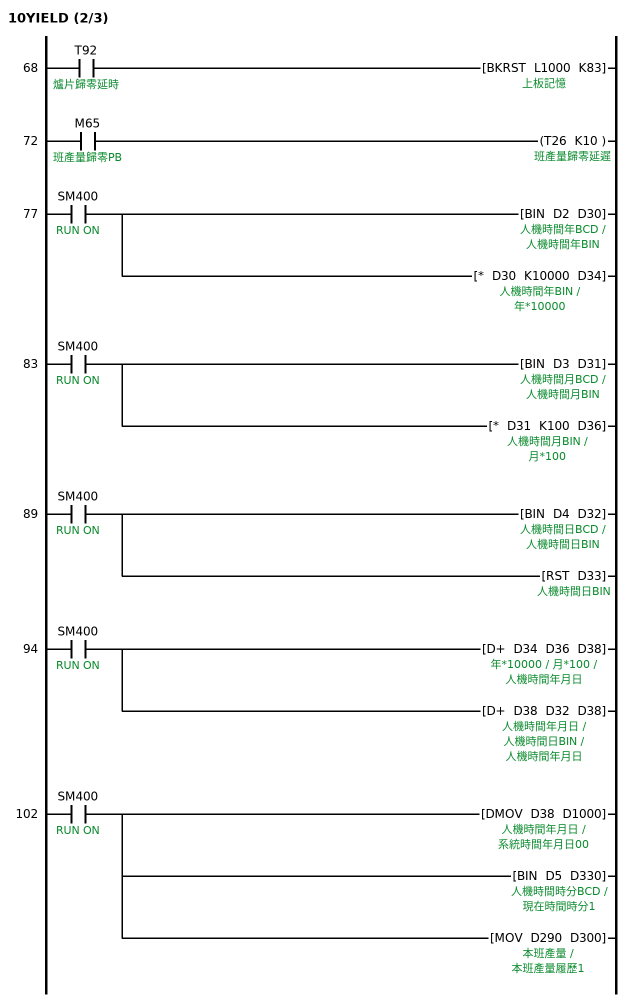
68    LD      T92  ; 爐片歸零延時
      BKRST   L1000 K83
72    LD      M65  ; 班產量歸零PB
      OUT     T26 K10  ; 班產量歸零延遲
77    LD      SM400  ; RUN ON
      BIN     D2 D30  ; 人機時間年BCD / 人機時間年BIN
      *       D30 K10000 D34  ; 年*10000
83    LD      SM400  ; RUN ON
      BIN     D3 D31  ; 人機時間月BCD / 人機時間月BIN
      *       D31 K100 D36  ; 月*100
89    LD      SM400  ; RUN ON
      BIN     D4 D32  ; 人機時間日BCD / 人機時間日BIN
      RST     D33  ; 人機時間日BIN
94    LD      SM400  ; RUN ON
      D+      D34 D36 D38  ; 人機時間年月日
      D+      D38 D32 D38
102   LD      SM400  ; RUN ON
      DMOV    D38 D1000  ; 系統時間年月日00
      BIN     D5 D330  ; 人機時間時分BCD / 現在時間時分1
      MOV     D290 D300  ; 本班產量履歷1
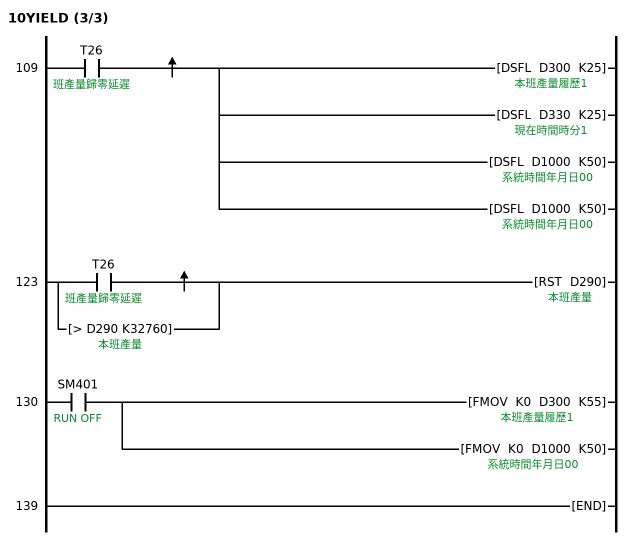
109   LD      T26  ; 班產量歸零延遲
      MEP
      DSFL    D300 K25
      DSFL    D330 K25
      DSFL    D1000 K50
      DSFL    D1000 K50
123   LD      T26  ; 班產量歸零延遲
      MEP
      OR>     D290 K32760  ; 本班產量
      RST     D290  ; 本班產量
130   LD      SM401  ; RUN OFF
      FMOV    K0 D300 K55
      FMOV    K0 D1000 K50
139   END
END_PROGRAM

PROGRAM 11MAINTE
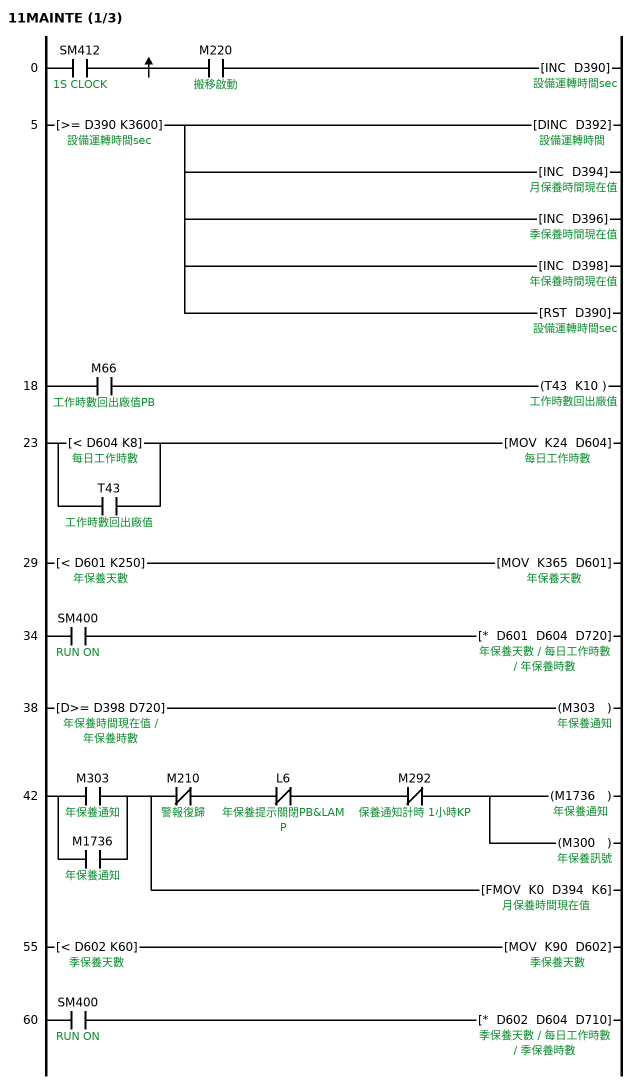
0     LD      SM412  ; 1S CLOCK
      MEP
      AND     M220  ; 搬移啟動
      INC     D390  ; 設備運轉時間sec
5     LD>=    D390 K3600  ; 設備運轉時間sec
      DINC    D392  ; 設備運轉時間
      INC     D394  ; 月保養時間現在值
      INC     D396  ; 季保養時間現在值
      INC     D398  ; 年保養時間現在值
      RST     D390  ; 設備運轉時間sec
18    LD      M66  ; 工作時數回出廠值PB
      OUT     T43 K10  ; 工作時數回出廠值
23    LD<     D604 K8  ; 每日工作時數
      OR      T43  ; 工作時數回出廠值
      MOV     K24 D604
29    LD<     D601 K250  ; 年保養天數
      MOV     K365 D601
34    LD      SM400  ; RUN ON
      *       D601 D604 D720  ; 年保養時數
38    LDD>=   D398 D720  ; 年保養時間現在值 / 年保養時數
      OUT     M303  ; 年保養通知
42    LD      M303  ; 年保養通知
      OR      M1736  ; 年保養通知
      MPS
      ANI     M210  ; 警報復歸
      ANI     L6  ; 年保養提示關閉PB&LAMP
      ANI     M292  ; 保養通知計時 1小時KP
      OUT     M1736  ; 年保養通知
      OUT     M300  ; 年保養訊號
      MPP
      FMOV    K0 D394 K6
55    LD<     D602 K60  ; 季保養天數
      MOV     K90 D602
60    LD      SM400  ; RUN ON
      *       D602 D604 D710  ; 季保養時數
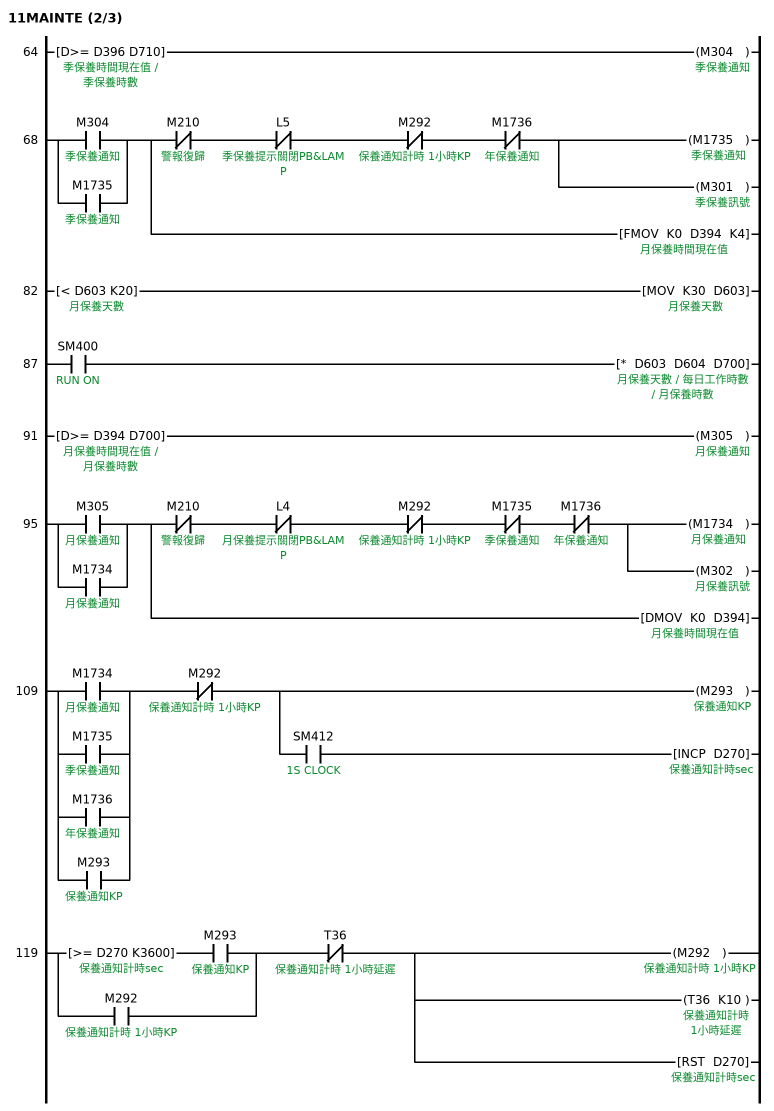
64    LDD>=   D396 D710  ; 季保養時間現在值 / 季保養時數
      OUT     M304  ; 季保養通知
68    LD      M304  ; 季保養通知
      OR      M1735  ; 季保養通知
      MPS
      ANI     M210  ; 警報復歸
      ANI     L5  ; 季保養提示關閉PB&LAMP
      ANI     M292  ; 保養通知計時 1小時KP
      ANI     M1736  ; 年保養通知
      OUT     M1735  ; 季保養通知
      OUT     M301  ; 季保養訊號
      MPP
      FMOV    K0 D394 K4
82    LD<     D603 K20  ; 月保養天數
      MOV     K30 D603
87    LD      SM400  ; RUN ON
      *       D603 D604 D700  ; 月保養時數
91    LDD>=   D394 D700  ; 月保養時間現在值 / 月保養時數
      OUT     M305  ; 月保養通知
95    LD      M305  ; 月保養通知
      OR      M1734  ; 月保養通知
      MPS
      ANI     M210  ; 警報復歸
      ANI     L4  ; 月保養提示關閉PB&LAMP
      ANI     M292  ; 保養通知計時 1小時KP
      ANI     M1735  ; 季保養通知
      ANI     M1736  ; 年保養通知
      OUT     M1734  ; 月保養通知
      OUT     M302  ; 月保養訊號
      MPP
      DMOV    K0 D394
109   LD      M1734  ; 月保養通知
      OR      M1735  ; 季保養通知
      OR      M1736  ; 年保養通知
      OR      M293  ; 保養通知KP
      ANI     M292  ; 保養通知計時 1小時KP
      OUT     M293  ; 保養通知KP
      AND     SM412  ; 1S CLOCK
      INCP    D270  ; 保養通知計時sec
119   LD>=    D270 K3600  ; 保養通知計時sec
      AND     M293  ; 保養通知KP
      OR      M292  ; 保養通知計時 1小時KP
      ANI     T36  ; 保養通知計時 1小時延遲
      OUT     M292  ; 保養通知計時 1小時KP
      OUT     T36 K10  ; 保養通知計時 1小時延遲
      RST     D270  ; 保養通知計時sec
